LIN {X 0,Y 144.028,Z 768.399,A -85,B 0,C 180,E1 -24191.511,E2 -24191.511} C_VEL
LIN {X 0,Y 142.223,Z 772.01,A -85,B 0,C 180,E1 -24195.698,E2 -24195.698} C_VEL
LIN {X 0,Y 141.401,Z 773.873,A -85,B 0,C 180,E1 -24198.535,E2 -24198.535} C_VEL
LIN {X 0,Y 140.849,Z 775.271,A -85,B 0,C 180,E1 -24201.394,E2 -24201.394} C_VEL
LIN {X 0,Y 140.554,Z 776.27,A -85,B 0,C 180,E1 -24204.263,E2 -24204.263} C_VEL
LIN {X 0,Y 140.569,Z 777.067,A -85,B 0,C 180,E1 -24209.359,E2 -24209.359} C_VEL
LIN {X 0,Y 140.705,Z 776.87,A -85,B 0,C 180,E1 -24212.866,E2 -24212.866} C_VEL
LIN {X 0,Y 141.078,Z 776.256,A -85,B 0,C 180,E1 -24215.721,E2 -24215.721} C_VEL
LIN {X 0,Y 142.6,Z 773.851,A -85,B 0,C 180,E1 -24221.372,E2 -24221.372} C_VEL
LIN {X 0,Y 144.414,Z 771.718,A -85,B 0,C 180,E1 -24224.805,E2 -24224.805} C_VEL
LIN {X 0,Y 147.56,Z 777.302,A -85,B 0,C 180,E1 -24230.931,E2 -24230.931} C_VEL
LIN {X 0,Y 150.794,Z 779.846,A -85,B 0,C 180,E1 -24234.803,E2 -24234.803} C_VEL
LIN {X 0,Y 153.542,Z 781.108,A -85,B 0,C 180,E1 -24237.243,E2 -24237.243} C_VEL
LIN {X 0,Y 156.869,Z 781.934,A -85,B 0,C 180,E1 -24239.528,E2 -24239.528} C_VEL
LIN {X 0,Y 164.35,Z 782.268,A -85,B 0,C 180,E1 -24243.776,E2 -24243.776} C_VEL
LIN {X 0,Y 168.6,Z 781.872,A -85,B 0,C 180,E1 -24245.705,E2 -24245.705} C_VEL
LIN {X 0,Y 173.147,Z 780.97,A -85,B 0,C 180,E1 -24247.508,E2 -24247.508} C_VEL
LIN {X 0,Y 182.916,Z 777.866,A -85,B 0,C 180,E1 -24250.784,E2 -24250.784} C_VEL
LIN {X 0,Y 190.879,Z 774.269,A -85,B 0,C 180,E1 -24252.936,E2 -24252.936} C_VEL
LIN {X 0,Y 199.307,Z 769.471,A -85,B 0,C 180,E1 -24254.851,E2 -24254.851} C_VEL
LIN {X 0,Y 203.849,Z 766.375,A -85,B 0,C 180,E1 -24255.76,E2 -24255.76} C_VEL
LIN {X 0,Y 203.147,Z 766.886,A -85,B 0,C 180,E1 -24256.218,E2 -24256.218} C_VEL
LIN {X 0,Y 194.513,Z 772.435,A -85,B 0,C 180,E1 -24258.054,E2 -24258.054} C_VEL
LIN {X 0,Y 186.285,Z 776.45,A -85,B 0,C 180,E1 -24260.107,E2 -24260.107} C_VEL
LIN {X 0,Y 181.112,Z 778.475,A -85,B 0,C 180,E1 -24261.62,E2 -24261.62} C_VEL
LIN {X 0,Y 176.183,Z 779.958,A -85,B 0,C 180,E1 -24263.248,E2 -24263.248} C_VEL
LIN {X 0,Y 171.503,Z 780.907,A -85,B 0,C 180,E1 -24264.991,E2 -24264.991} C_VEL
LIN {X 0,Y 167.024,Z 781.435,A -85,B 0,C 180,E1 -24266.838,E2 -24266.838} C_VEL
LIN {X 0,Y 162.831,Z 781.546,A -85,B 0,C 180,E1 -24268.806,E2 -24268.806} C_VEL
LIN {X 0,Y 159.015,Z 781.191,A -85,B 0,C 180,E1 -24270.911,E2 -24270.911} C_VEL
LIN {X 0,Y 155.536,Z 780.325,A -85,B 0,C 180,E1 -24273.137,E2 -24273.137} C_VEL
LIN {X 0,Y 152.482,Z 779.046,A -85,B 0,C 180,E1 -24275.492,E2 -24275.492} C_VEL
LIN {X 0,Y 148.803,Z 776.375,A -85,B 0,C 180,E1 -24279.254,E2 -24279.254} C_VEL
LIN {X 0,Y 146.088,Z 772.671,A -85,B 0,C 180,E1 -24283.223,E2 -24283.223} C_VEL
LIN {X 0,Y 144.244,Z 767.118,A -85,B 0,C 180,E1 -24287.917,E2 -24287.917} C_VEL
LIN {X 0,Y 143.675,Z 760.498,A -85,B 0,C 180,E1 -24292.269,E2 -24292.269} C_VEL
LIN {X 0,Y 143.884,Z 753.954,A -85,B 0,C 180,E1 -24295.798,E2 -24295.798} C_VEL
LIN {X 0,Y 144.25,Z 747.49,A -85,B 0,C 180,E1 -24298.604,E2 -24298.604} C_VEL
LIN {X 0,Y 144.568,Z 738.067,A -85,B 0,C 180,E1 -24301.741,E2 -24301.741} C_VEL
LIN {X 0,Y 144.815,Z 730.254,A -85,B 0,C 180,E1 -24303.826,E2 -24303.826} C_VEL
LIN {X 0,Y 145.107,Z 718.487,A -85,B 0,C 180,E1 -24306.256,E2 -24306.256} C_VEL
LIN {X 0,Y 145.333,Z 708.147,A -85,B 0,C 180,E1 -24307.817,E2 -24307.817} C_VEL
LIN {X 0,Y 145.44,Z 690.055,A -85,B 0,C 180,E1 -24309.737,E2 -24309.737} C_VEL
LIN {X 0,Y 145.416,Z 656.523,A -85,B 0,C 180,E1 -24313.05,E2 -24313.05} C_VEL
LIN {X 0,Y 143.902,Z 632.91,A -85,B 0,C 180,E1 -24315.219,E2 -24315.219} C_VEL
LIN {X 0,Y 143.753,Z 627.443,A -85,B 0,C 180,E1 -24317.058,E2 -24317.058} C_VEL
LIN {X 0,Y 145.393,Z 608.667,A -85,B 0,C 180,E1 -24323.842,E2 -24323.842} C_VEL
LIN {X 0,Y 145.884,Z 605.68,A -85,B 0,C 180,E1 -24325.312,E2 -24325.312} C_VEL
LIN {X 0,Y 146.21,Z 605.142,A -85,B 0,C 180,E1 -24326.016,E2 -24326.016} C_VEL
LIN {X 0,Y 147.642,Z 604.988,A -85,B 0,C 180,E1 -24327.269,E2 -24327.269} C_VEL
LIN {X 0,Y 149.873,Z 603.29,A -85,B 0,C 180,E1 -24328.728,E2 -24328.728} C_VEL
LIN {X 0,Y 154.133,Z 597.997,A -85,B 0,C 180,E1 -24331.052,E2 -24331.052} C_VEL
LIN {X 0,Y 154.864,Z 597.508,A -85,B 0,C 180,E1 -24331.459,E2 -24331.459} C_VEL
LIN {X 0,Y 157.666,Z 597.465,A -85,B 0,C 180,E1 -24333.097,E2 -24333.097} C_VEL
LIN {X 0,Y 159.705,Z 596.432,A -85,B 0,C 180,E1 -24334.131,E2 -24334.131} C_VEL
LIN {X 0,Y 164.294,Z 595.958,A -85,B 0,C 180,E1 -24336.408,E2 -24336.408} C_VEL
LIN {X 0,Y 165.416,Z 595.863,A -85,B 0,C 180,E1 -24336.93,E2 -24336.93} C_VEL
LIN {X 0,Y 171.993,Z 606.336,A -85,B 0,C 180,E1 -24340.443,E2 -24340.443} C_VEL
LIN {X 0,Y 177.72,Z 616.812,A -85,B 0,C 180,E1 -24343.192,E2 -24343.192} C_VEL
LIN {X 0,Y 180.855,Z 624.587,A -85,B 0,C 180,E1 -24344.681,E2 -24344.681} C_VEL
LIN {X 0,Y 178.029,Z 666.301,A -85,B 0,C 180,E1 -24346.194,E2 -24346.194} C_VEL
LIN {X 0,Y 176.211,Z 679.252,A -85,B 0,C 180,E1 -24347.012,E2 -24347.012} C_VEL
LIN {X 0,Y 173.885,Z 691.223,A -85,B 0,C 180,E1 -24348.17,E2 -24348.17} C_VEL
LIN {X 0,Y 170.991,Z 702.495,A -85,B 0,C 180,E1 -24349.656,E2 -24349.656} C_VEL
LIN {X 0,Y 167.18,Z 714.119,A -85,B 0,C 180,E1 -24351.676,E2 -24351.676} C_VEL
LIN {X 0,Y 163.151,Z 724.561,A -85,B 0,C 180,E1 -24354.059,E2 -24354.059} C_VEL
LIN {X 0,Y 159.522,Z 733.089,A -85,B 0,C 180,E1 -24356.584,E2 -24356.584} C_VEL
LIN {X 0,Y 155.782,Z 741.183,A -85,B 0,C 180,E1 -24359.624,E2 -24359.624} C_VEL
LIN {X 0,Y 151.851,Z 748.611,A -85,B 0,C 180,E1 -24363.173,E2 -24363.173} C_VEL
LIN {X 0,Y 147.83,Z 755.661,A -85,B 0,C 180,E1 -24367.643,E2 -24367.643} C_VEL
LIN {X 0,Y 145.189,Z 760.348,A -85,B 0,C 180,E1 -24371.659,E2 -24371.659} C_VEL
LIN {X 0,Y 143.132,Z 763.929,A -85,B 0,C 180,E1 -24375.786,E2 -24375.786} C_VEL
LIN {X 0,Y 142.14,Z 765.777,A -85,B 0,C 180,E1 -24378.59,E2 -24378.59} C_VEL
LIN {X 0,Y 141.435,Z 767.165,A -85,B 0,C 180,E1 -24381.424,E2 -24381.424} C_VEL
LIN {X 0,Y 141.008,Z 768.151,A -85,B 0,C 180,E1 -24384.277,E2 -24384.277} C_VEL
LIN {X 0,Y 140.737,Z 768.758,A -85,B 0,C 180,E1 -24387.135,E2 -24387.135} C_VEL
LIN {X 0,Y 140.69,Z 768.984,A -85,B 0,C 180,E1 -24389.997,E2 -24389.997} C_VEL
LIN {X 0,Y 140.736,Z 768.789,A -85,B 0,C 180,E1 -24392.86,E2 -24392.86} C_VEL
LIN {X 0,Y 141.007,Z 768.204,A -85,B 0,C 180,E1 -24395.718,E2 -24395.718} C_VEL
LIN {X 0,Y 142.136,Z 765.884,A -85,B 0,C 180,E1 -24401.405,E2 -24401.405} C_VEL
LIN {X 0,Y 143.73,Z 763.013,A -85,B 0,C 180,E1 -24405.598,E2 -24405.598} C_VEL
LIN {X 0,Y 145.977,Z 759.117,A -85,B 0,C 180,E1 -24409.692,E2 -24409.692} C_VEL
LIN {X 0,Y 148.832,Z 754.096,A -85,B 0,C 180,E1 -24413.662,E2 -24413.662} C_VEL
LIN {X 0,Y 152.426,Z 747.763,A -85,B 0,C 180,E1 -24417.454,E2 -24417.454} C_VEL
LIN {X 0,Y 156.142,Z 740.567,A -85,B 0,C 180,E1 -24420.801,E2 -24420.801} C_VEL
LIN {X 0,Y 160.208,Z 731.769,A -85,B 0,C 180,E1 -24424.005,E2 -24424.005} C_VEL
LIN {X 0,Y 164.355,Z 721.911,A -85,B 0,C 180,E1 -24426.771,E2 -24426.771} C_VEL
LIN {X 0,Y 168.491,Z 710.804,A -85,B 0,C 180,E1 -24429.112,E2 -24429.112} C_VEL
LIN {X 0,Y 171.827,Z 699.911,A -85,B 0,C 180,E1 -24430.873,E2 -24430.873} C_VEL
LIN {X 0,Y 174.767,Z 687.858,A -85,B 0,C 180,E1 -24432.341,E2 -24432.341} C_VEL
LIN {X 0,Y 177.064,Z 675.297,A -85,B 0,C 180,E1 -24433.417,E2 -24433.417} C_VEL
LIN {X 0,Y 178.617,Z 661.534,A -85,B 0,C 180,E1 -24434.161,E2 -24434.161} C_VEL
LIN {X 0,Y 181.017,Z 624.783,A -85,B 0,C 180,E1 -24435.451,E2 -24435.451} C_VEL
LIN {X 0,Y 177.262,Z 615.771,A -85,B 0,C 180,E1 -24437.232,E2 -24437.232} C_VEL
LIN {X 0,Y 171.653,Z 605.747,A -85,B 0,C 180,E1 -24439.947,E2 -24439.947} C_VEL
LIN {X 0,Y 166.095,Z 596.95,A -85,B 0,C 180,E1 -24442.917,E2 -24442.917} C_VEL
LIN {X 0,Y 161.752,Z 590.626,A -85,B 0,C 180,E1 -24445.502,E2 -24445.502} C_VEL
LIN {X 0,Y 159.087,Z 586.943,A -85,B 0,C 180,E1 -24447.236,E2 -24447.236} C_VEL
LIN {X 0,Y 156.431,Z 583.247,A -85,B 0,C 180,E1 -24449.115,E2 -24449.115} C_VEL
LIN {X 0,Y 153.386,Z 579.693,A -85,B 0,C 180,E1 -24451.429,E2 -24451.429} C_VEL
LIN {X 0,Y 152.306,Z 577.95,A -85,B 0,C 180,E1 -24452.364,E2 -24452.364} C_VEL
LIN {X 0,Y 149.696,Z 575.629,A -85,B 0,C 180,E1 -24454.609,E2 -24454.609} C_VEL
LIN {X 0,Y 148.169,Z 572.836,A -85,B 0,C 180,E1 -24456.223,E2 -24456.223} C_VEL
LIN {X 0,Y 147.867,Z 572.413,A -85,B 0,C 180,E1 -24456.543,E2 -24456.543} C_VEL
LIN {X 0,Y 145.469,Z 570.904,A -85,B 0,C 180,E1 -24459.052,E2 -24459.052} C_VEL
LIN {X 0,Y 143.832,Z 568.536,A -85,B 0,C 180,E1 -24461.205,E2 -24461.205} C_VEL
LIN {X 0,Y 143.277,Z 566.62,A -85,B 0,C 180,E1 -24462.331,E2 -24462.331} C_VEL
LIN {X 0,Y 143.588,Z 566.58,A -85,B 0,C 180,E1 -24468.709,E2 -24468.709} C_VEL
LIN {X 0,Y 143.658,Z 566.571,A -85,B 0,C 180,E1 -24471.56,E2 -24471.56} C_VEL
LIN {X 0,Y 144.172,Z 566.526,A -85,B 0,C 180,E1 -24480,E2 -24480} C_VEL
LIN {X 0,Y 143.678,Z 566.573,A -85,B 0,C 180,E1 -24488.438,E2 -24488.438} C_VEL
LIN {X 0,Y 143.565,Z 566.586,A -85,B 0,C 180,E1 -24491.758,E2 -24491.758} C_VEL
LIN {X 0,Y 143.287,Z 566.712,A -85,B 0,C 180,E1 -24497.483,E2 -24497.483} C_VEL
LIN {X 0,Y 143.993,Z 568.912,A -85,B 0,C 180,E1 -24498.681,E2 -24498.681} C_VEL
LIN {X 0,Y 145.834,Z 571.244,A -85,B 0,C 180,E1 -24501.008,E2 -24501.008} C_VEL
LIN {X 0,Y 148.092,Z 572.648,A -85,B 0,C 180,E1 -24503.326,E2 -24503.326} C_VEL
LIN {X 0,Y 149.662,Z 575.61,A -85,B 0,C 180,E1 -24505.001,E2 -24505.001} C_VEL
LIN {X 0,Y 152.591,Z 578.318,A -85,B 0,C 180,E1 -24507.517,E2 -24507.517} C_VEL
LIN {X 0,Y 154.86,Z 581.681,A -85,B 0,C 180,E1 -24509.387,E2 -24509.387} C_VEL
LIN {X 0,Y 156.547,Z 583.503,A -85,B 0,C 180,E1 -24510.618,E2 -24510.618} C_VEL
LIN {X 0,Y 159.281,Z 587.171,A -85,B 0,C 180,E1 -24512.531,E2 -24512.531} C_VEL
LIN {X 0,Y 161.27,Z 590.154,A -85,B 0,C 180,E1 -24513.848,E2 -24513.848} C_VEL
LIN {X 0,Y 165.359,Z 596.983,A -85,B 0,C 180,E1 -24516.384,E2 -24516.384} C_VEL
LIN {X 0,Y 170.544,Z 606.854,A -85,B 0,C 180,E1 -24519.316,E2 -24519.316} C_VEL
LIN {X 0,Y 175.217,Z 617.057,A -85,B 0,C 180,E1 -24521.752,E2 -24521.752} C_VEL
LIN {X 0,Y 179.914,Z 629.167,A -85,B 0,C 180,E1 -24524.074,E2 -24524.074} C_VEL
LIN {X 0,Y 180.657,Z 631.54,A -85,B 0,C 180,E1 -24524.447,E2 -24524.447} C_VEL
LIN {X 0,Y 177.79,Z 673.247,A -85,B 0,C 180,E1 -24525.933,E2 -24525.933} C_VEL
LIN {X 0,Y 175.882,Z 686.736,A -85,B 0,C 180,E1 -24526.773,E2 -24526.773} C_VEL
LIN {X 0,Y 173.121,Z 699.519,A -85,B 0,C 180,E1 -24527.949,E2 -24527.949} C_VEL
LIN {X 0,Y 170.042,Z 710.602,A -85,B 0,C 180,E1 -24529.389,E2 -24529.389} C_VEL
LIN {X 0,Y 166.132,Z 722.153,A -85,B 0,C 180,E1 -24531.396,E2 -24531.396} C_VEL
LIN {X 0,Y 162.027,Z 732.557,A -85,B 0,C 180,E1 -24533.776,E2 -24533.776} C_VEL
LIN {X 0,Y 158.192,Z 741.068,A -85,B 0,C 180,E1 -24536.269,E2 -24536.269} C_VEL
LIN {X 0,Y 154.4,Z 748.922,A -85,B 0,C 180,E1 -24539.201,E2 -24539.201} C_VEL
LIN {X 0,Y 150.544,Z 756.602,A -85,B 0,C 180,E1 -24542.927,E2 -24542.927} C_VEL
LIN {X 0,Y 147.137,Z 762.745,A -85,B 0,C 180,E1 -24546.772,E2 -24546.772} C_VEL
LIN {X 0,Y 145.111,Z 765.37,A -85,B 0,C 180,E1 -24548.7,E2 -24548.7} C_VEL
LIN {X 0,Y 140.306,Z 769.068,A -85,B 0,C 180,E1 -24551.862,E2 -24551.862} C_VEL
LIN {X 0,Y 136.608,Z 771.488,A -85,B 0,C 180,E1 -24554.599,E2 -24554.599} C_VEL
LIN {X 0,Y 134.793,Z 773.041,A -85,B 0,C 180,E1 -24556.879,E2 -24556.879} C_VEL
LIN {X 0,Y 134.497,Z 773.51,A -85,B 0,C 180,E1 -24557.678,E2 -24557.678} C_VEL
LIN {X 0,Y 133.823,Z 775.066,A -85,B 0,C 180,E1 -24560.938,E2 -24560.938} C_VEL
LIN {X 0,Y 133.397,Z 776.676,A -85,B 0,C 180,E1 -24566.983,E2 -24566.983} C_VEL
LIN {X 0,Y 133.532,Z 776.891,A -85,B 0,C 180,E1 -24570.003,E2 -24570.003} C_VEL
LIN {X 0,Y 134.028,Z 776.052,A -85,B 0,C 180,E1 -24576.023,E2 -24576.023} C_VEL
LIN {X 0,Y 135.653,Z 773.646,A -85,B 0,C 180,E1 -24581.963,E2 -24581.963} C_VEL
LIN {X 0,Y 138.304,Z 770.641,A -85,B 0,C 180,E1 -24586.611,E2 -24586.611} C_VEL
LIN {X 0,Y 141.148,Z 775.592,A -85,B 0,C 180,E1 -24591.93,E2 -24591.93} C_VEL
LIN {X 0,Y 144.491,Z 778.609,A -85,B 0,C 180,E1 -24595.963,E2 -24595.963} C_VEL
LIN {X 0,Y 147.354,Z 780.07,A -85,B 0,C 180,E1 -24598.489,E2 -24598.489} C_VEL
LIN {X 0,Y 154.444,Z 781.964,A -85,B 0,C 180,E1 -24603.1,E2 -24603.1} C_VEL
LIN {X 0,Y 158.507,Z 782.227,A -85,B 0,C 180,E1 -24605.201,E2 -24605.201} C_VEL
LIN {X 0,Y 162.885,Z 782.108,A -85,B 0,C 180,E1 -24607.163,E2 -24607.163} C_VEL
LIN {X 0,Y 167.589,Z 781.623,A -85,B 0,C 180,E1 -24608.982,E2 -24608.982} C_VEL
LIN {X 0,Y 172.532,Z 780.703,A -85,B 0,C 180,E1 -24610.676,E2 -24610.676} C_VEL
LIN {X 0,Y 177.661,Z 779.286,A -85,B 0,C 180,E1 -24612.262,E2 -24612.262} C_VEL
LIN {X 0,Y 185.853,Z 776.369,A -85,B 0,C 180,E1 -24614.395,E2 -24614.395} C_VEL
LIN {X 0,Y 189.989,Z 774.505,A -85,B 0,C 180,E1 -24615.344,E2 -24615.344} C_VEL
LIN {X 0,Y 192.289,Z 773.406,A -85,B 0,C 180,E1 -24616.018,E2 -24616.018} C_VEL
LIN {X 0,Y 183.718,Z 777.157,A -85,B 0,C 180,E1 -24617.975,E2 -24617.975} C_VEL
LIN {X 0,Y 175.648,Z 779.743,A -85,B 0,C 180,E1 -24620.194,E2 -24620.194} C_VEL
LIN {X 0,Y 166.894,Z 781.396,A -85,B 0,C 180,E1 -24623.143,E2 -24623.143} C_VEL
LIN {X 0,Y 161.119,Z 781.691,A -85,B 0,C 180,E1 -24625.455,E2 -24625.455} C_VEL
LIN {X 0,Y 156.808,Z 781.382,A -85,B 0,C 180,E1 -24627.464,E2 -24627.464} C_VEL
LIN {X 0,Y 152.879,Z 780.647,A -85,B 0,C 180,E1 -24629.623,E2 -24629.623} C_VEL
LIN {X 0,Y 149.294,Z 779.53,A -85,B 0,C 180,E1 -24631.917,E2 -24631.917} C_VEL
LIN {X 0,Y 144.767,Z 777.023,A -85,B 0,C 180,E1 -24635.629,E2 -24635.629} C_VEL
LIN {X 0,Y 141.32,Z 773.548,A -85,B 0,C 180,E1 -24639.628,E2 -24639.628} C_VEL
LIN {X 0,Y 138.685,Z 768.495,A -85,B 0,C 180,E1 -24644.341,E2 -24644.341} C_VEL
LIN {X 0,Y 137.443,Z 762.266,A -85,B 0,C 180,E1 -24648.945,E2 -24648.945} C_VEL
LIN {X 0,Y 137.312,Z 756.216,A -85,B 0,C 180,E1 -24652.649,E2 -24652.649} C_VEL
LIN {X 0,Y 137.636,Z 748.736,A -85,B 0,C 180,E1 -24656.341,E2 -24656.341} C_VEL
LIN {X 0,Y 137.901,Z 741.278,A -85,B 0,C 180,E1 -24659.27,E2 -24659.27} C_VEL
LIN {X 0,Y 138.187,Z 733.012,A -85,B 0,C 180,E1 -24661.822,E2 -24661.822} C_VEL
LIN {X 0,Y 138.339,Z 723.891,A -85,B 0,C 180,E1 -24664.006,E2 -24664.006} C_VEL
LIN {X 0,Y 138.591,Z 713.294,A -85,B 0,C 180,E1 -24666.004,E2 -24666.004} C_VEL
LIN {X 0,Y 138.742,Z 700.731,A -85,B 0,C 180,E1 -24667.641,E2 -24667.641} C_VEL
LIN {X 0,Y 138.647,Z 657.852,A -85,B 0,C 180,E1 -24672.236,E2 -24672.236} C_VEL
LIN {X 0,Y 136.908,Z 632.582,A -85,B 0,C 180,E1 -24674.7,E2 -24674.7} C_VEL
LIN {X 0,Y 136.728,Z 626.035,A -85,B 0,C 180,E1 -24677.191,E2 -24677.191} C_VEL
LIN {X 0,Y 137.028,Z 622.984,A -85,B 0,C 180,E1 -24678.891,E2 -24678.891} C_VEL
LIN {X 0,Y 137.175,Z 622.556,A -85,B 0,C 180,E1 -24679.452,E2 -24679.452} C_VEL
LIN {X 0,Y 138.377,Z 622.348,A -85,B 0,C 180,E1 -24681.015,E2 -24681.015} C_VEL
LIN {X 0,Y 140.519,Z 619.897,A -85,B 0,C 180,E1 -24682.889,E2 -24682.889} C_VEL
LIN {X 0,Y 145.658,Z 612.31,A -85,B 0,C 180,E1 -24686.508,E2 -24686.508} C_VEL
LIN {X 0,Y 148.347,Z 611.466,A -85,B 0,C 180,E1 -24688.454,E2 -24688.454} C_VEL
LIN {X 0,Y 151.116,Z 609.222,A -85,B 0,C 180,E1 -24690.143,E2 -24690.143} C_VEL
LIN {X 0,Y 155.04,Z 604.642,A -85,B 0,C 180,E1 -24692.184,E2 -24692.184} C_VEL
LIN {X 0,Y 157.427,Z 604.468,A -85,B 0,C 180,E1 -24693.536,E2 -24693.536} C_VEL
LIN {X 0,Y 159.975,Z 603.536,A -85,B 0,C 180,E1 -24694.828,E2 -24694.828} C_VEL
LIN {X 0,Y 163.435,Z 603.345,A -85,B 0,C 180,E1 -24696.535,E2 -24696.535} C_VEL
LIN {X 0,Y 168.981,Z 612.485,A -85,B 0,C 180,E1 -24699.625,E2 -24699.625} C_VEL
LIN {X 0,Y 173.751,Z 621.62,A -85,B 0,C 180,E1 -24702.06,E2 -24702.06} C_VEL
LIN {X 0,Y 175.803,Z 626.867,A -85,B 0,C 180,E1 -24703.112,E2 -24703.112} C_VEL
LIN {X 0,Y 172.998,Z 666.342,A -85,B 0,C 180,E1 -24704.558,E2 -24704.558} C_VEL
LIN {X 0,Y 171.072,Z 679.645,A -85,B 0,C 180,E1 -24705.41,E2 -24705.41} C_VEL
LIN {X 0,Y 168.411,Z 692.512,A -85,B 0,C 180,E1 -24706.686,E2 -24706.686} C_VEL
LIN {X 0,Y 165.161,Z 704.285,A -85,B 0,C 180,E1 -24708.324,E2 -24708.324} C_VEL
LIN {X 0,Y 161.198,Z 715.615,A -85,B 0,C 180,E1 -24710.382,E2 -24710.382} C_VEL
LIN {X 0,Y 157.04,Z 725.823,A -85,B 0,C 180,E1 -24712.829,E2 -24712.829} C_VEL
LIN {X 0,Y 152.807,Z 734.979,A -85,B 0,C 180,E1 -24715.706,E2 -24715.706} C_VEL
LIN {X 0,Y 148.332,Z 743.875,A -85,B 0,C 180,E1 -24719.378,E2 -24719.378} C_VEL
LIN {X 0,Y 144.284,Z 751.036,A -85,B 0,C 180,E1 -24723.218,E2 -24723.218} C_VEL
LIN {X 0,Y 141.28,Z 755.868,A -85,B 0,C 180,E1 -24726.547,E2 -24726.547} C_VEL
LIN {X 0,Y 138.469,Z 760.554,A -85,B 0,C 180,E1 -24730.734,E2 -24730.734} C_VEL
LIN {X 0,Y 136.246,Z 764.135,A -85,B 0,C 180,E1 -24735.051,E2 -24735.051} C_VEL
LIN {X 0,Y 135.175,Z 765.983,A -85,B 0,C 180,E1 -24737.994,E2 -24737.994} C_VEL
LIN {X 0,Y 134.429,Z 767.369,A -85,B 0,C 180,E1 -24740.974,E2 -24740.974} C_VEL
LIN {X 0,Y 133.95,Z 768.356,A -85,B 0,C 180,E1 -24743.974,E2 -24743.974} C_VEL
LIN {X 0,Y 133.596,Z 769.099,A -85,B 0,C 180,E1 -24748.24,E2 -24748.24} C_VEL
LIN {X 0,Y 133.659,Z 768.993,A -85,B 0,C 180,E1 -24753.011,E2 -24753.011} C_VEL
LIN {X 0,Y 133.948,Z 768.409,A -85,B 0,C 180,E1 -24756.021,E2 -24756.021} C_VEL
LIN {X 0,Y 135.171,Z 766.089,A -85,B 0,C 180,E1 -24762.001,E2 -24762.001} C_VEL
LIN {X 0,Y 136.901,Z 763.217,A -85,B 0,C 180,E1 -24766.398,E2 -24766.398} C_VEL
LIN {X 0,Y 139.306,Z 759.321,A -85,B 0,C 180,E1 -24770.677,E2 -24770.677} C_VEL
LIN {X 0,Y 142.347,Z 754.299,A -85,B 0,C 180,E1 -24774.81,E2 -24774.81} C_VEL
LIN {X 0,Y 146.163,Z 747.966,A -85,B 0,C 180,E1 -24778.737,E2 -24778.737} C_VEL
LIN {X 0,Y 150.678,Z 739.542,A -85,B 0,C 180,E1 -24782.705,E2 -24782.705} C_VEL
LIN {X 0,Y 155.218,Z 730.194,A -85,B 0,C 180,E1 -24786.056,E2 -24786.056} C_VEL
LIN {X 0,Y 159.665,Z 719.838,A -85,B 0,C 180,E1 -24788.844,E2 -24788.844} C_VEL
LIN {X 0,Y 164.043,Z 708.159,A -85,B 0,C 180,E1 -24791.198,E2 -24791.198} C_VEL
LIN {X 0,Y 167.56,Z 696.486,A -85,B 0,C 180,E1 -24792.964,E2 -24792.964} C_VEL
LIN {X 0,Y 170.383,Z 684.338,A -85,B 0,C 180,E1 -24794.315,E2 -24794.315} C_VEL
LIN {X 0,Y 172.602,Z 671.307,A -85,B 0,C 180,E1 -24795.308,E2 -24795.308} C_VEL
LIN {X 0,Y 173.916,Z 657.301,A -85,B 0,C 180,E1 -24795.964,E2 -24795.964} C_VEL
LIN {X 0,Y 175.972,Z 627.04,A -85,B 0,C 180,E1 -24797.024,E2 -24797.024} C_VEL
LIN {X 0,Y 172.81,Z 619.484,A -85,B 0,C 180,E1 -24798.633,E2 -24798.633} C_VEL
LIN {X 0,Y 167.634,Z 610.173,A -85,B 0,C 180,E1 -24801.322,E2 -24801.322} C_VEL
LIN {X 0,Y 162.011,Z 600.921,A -85,B 0,C 180,E1 -24804.586,E2 -24804.586} C_VEL
LIN {X 0,Y 156.679,Z 593.19,A -85,B 0,C 180,E1 -24808.103,E2 -24808.103} C_VEL
LIN {X 0,Y 153.194,Z 588.56,A -85,B 0,C 180,E1 -24810.714,E2 -24810.714} C_VEL
LIN {X 0,Y 150.501,Z 584.839,A -85,B 0,C 180,E1 -24812.995,E2 -24812.995} C_VEL
LIN {X 0,Y 147.145,Z 581.167,A -85,B 0,C 180,E1 -24816.141,E2 -24816.141} C_VEL
LIN {X 0,Y 146.081,Z 579.156,A -85,B 0,C 180,E1 -24817.363,E2 -24817.363} C_VEL
LIN {X 0,Y 143.353,Z 576.977,A -85,B 0,C 180,E1 -24820.489,E2 -24820.489} C_VEL
LIN {X 0,Y 141.734,Z 573.899,A -85,B 0,C 180,E1 -24822.97,E2 -24822.97} C_VEL
LIN {X 0,Y 141.469,Z 573.476,A -85,B 0,C 180,E1 -24823.402,E2 -24823.402} C_VEL
LIN {X 0,Y 138.7,Z 571.786,A -85,B 0,C 180,E1 -24828.306,E2 -24828.306} C_VEL
LIN {X 0,Y 136.736,Z 568.099,A -85,B 0,C 180,E1 -24835.578,E2 -24835.578} C_VEL
LIN {X 0,Y 136.722,Z 567.429,A -85,B 0,C 180,E1 -24836.685,E2 -24836.685} C_VEL
LIN {X 0,Y 137.129,Z 567.403,A -85,B 0,C 180,E1 -24840,E2 -24840} C_VEL
LIN {X 0,Y 136.712,Z 567.539,A -85,B 0,C 180,E1 -24843.5,E2 -24843.5} C_VEL
LIN {X 0,Y 137.235,Z 569.712,A -85,B 0,C 180,E1 -24846.986,E2 -24846.986} C_VEL
LIN {X 0,Y 140.336,Z 573.047,A -85,B 0,C 180,E1 -24854.501,E2 -24854.501} C_VEL
LIN {X 0,Y 141.681,Z 573.747,A -85,B 0,C 180,E1 -24856.572,E2 -24856.572} C_VEL
LIN {X 0,Y 143.097,Z 576.625,A -85,B 0,C 180,E1 -24858.803,E2 -24858.803} C_VEL
LIN {X 0,Y 145.486,Z 578.849,A -85,B 0,C 180,E1 -24861.663,E2 -24861.663} C_VEL
LIN {X 0,Y 146.238,Z 579.437,A -85,B 0,C 180,E1 -24862.46,E2 -24862.46} C_VEL
LIN {X 0,Y 148.311,Z 582.736,A -85,B 0,C 180,E1 -24864.683,E2 -24864.683} C_VEL
LIN {X 0,Y 150.439,Z 584.807,A -85,B 0,C 180,E1 -24866.594,E2 -24866.594} C_VEL
LIN {X 0,Y 153.062,Z 588.426,A -85,B 0,C 180,E1 -24868.824,E2 -24868.824} C_VEL
LIN {X 0,Y 154.391,Z 590.164,A -85,B 0,C 180,E1 -24869.86,E2 -24869.86} C_VEL
LIN {X 0,Y 157.717,Z 594.697,A -85,B 0,C 180,E1 -24872.267,E2 -24872.267} C_VEL
LIN {X 0,Y 162.367,Z 602.859,A -85,B 0,C 180,E1 -24875.376,E2 -24875.376} C_VEL
LIN {X 0,Y 167.211,Z 612.47,A -85,B 0,C 180,E1 -24878.291,E2 -24878.291} C_VEL
LIN {X 0,Y 171.382,Z 622.025,A -85,B 0,C 180,E1 -24880.617,E2 -24880.617} C_VEL
LIN {X 0,Y 175.614,Z 633.499,A -85,B 0,C 180,E1 -24882.87,E2 -24882.87} C_VEL
LIN {X 0,Y 172.714,Z 673.501,A -85,B 0,C 180,E1 -24884.321,E2 -24884.321} C_VEL
LIN {X 0,Y 170.734,Z 686.804,A -85,B 0,C 180,E1 -24885.163,E2 -24885.163} C_VEL
LIN {X 0,Y 167.93,Z 699.322,A -85,B 0,C 180,E1 -24886.331,E2 -24886.331} C_VEL
LIN {X 0,Y 164.716,Z 710.402,A -85,B 0,C 180,E1 -24887.781,E2 -24887.781} C_VEL
LIN {X 0,Y 160.625,Z 721.951,A -85,B 0,C 180,E1 -24889.81,E2 -24889.81} C_VEL
LIN {X 0,Y 156.337,Z 732.355,A -85,B 0,C 180,E1 -24892.233,E2 -24892.233} C_VEL
LIN {X 0,Y 152.333,Z 740.866,A -85,B 0,C 180,E1 -24894.785,E2 -24894.785} C_VEL
LIN {X 0,Y 148.323,Z 748.719,A -85,B 0,C 180,E1 -24897.791,E2 -24897.791} C_VEL
LIN {X 0,Y 144.216,Z 756.4,A -85,B 0,C 180,E1 -24901.636,E2 -24901.636} C_VEL
LIN {X 0,Y 140.066,Z 763.48,A -85,B 0,C 180,E1 -24906.337,E2 -24906.337} C_VEL
LIN {X 0,Y 137.28,Z 768.194,A -85,B 0,C 180,E1 -24910.566,E2 -24910.566} C_VEL
LIN {X 0,Y 135.33,Z 771.806,A -85,B 0,C 180,E1 -24914.953,E2 -24914.953} C_VEL
LIN {X 0,Y 134.497,Z 773.51,A -85,B 0,C 180,E1 -24917.678,E2 -24917.678} C_VEL
LIN {X 0,Y 133.339,Z 774.824,A -85,B 0,C 180,E1 -24920.089,E2 -24920.089} C_VEL
LIN {X 0,Y 131.45,Z 775.762,A -85,B 0,C 180,E1 -24922.493,E2 -24922.493} C_VEL
LIN {X 0,Y 127.514,Z 776.645,A -85,B 0,C 180,E1 -24927.488,E2 -24927.488} C_VEL
LIN {X 0,Y 126.493,Z 776.685,A -85,B 0,C 180,E1 -24930.147,E2 -24930.147} C_VEL
LIN {X 0,Y 126.427,Z 776.612,A -85,B 0,C 180,E1 -24931.049,E2 -24931.049} C_VEL
LIN {X 0,Y 126.974,Z 775.847,A -85,B 0,C 180,E1 -24936.358,E2 -24936.358} C_VEL
LIN {X 0,Y 128.736,Z 773.441,A -85,B 0,C 180,E1 -24942.616,E2 -24942.616} C_VEL
LIN {X 0,Y 132.057,Z 769.625,A -85,B 0,C 180,E1 -24948.223,E2 -24948.223} C_VEL
LIN {X 0,Y 132.594,Z 769.669,A -85,B 0,C 180,E1 -24948.947,E2 -24948.947} C_VEL
LIN {X 0,Y 135.91,Z 774.849,A -85,B 0,C 180,E1 -24954.439,E2 -24954.439} C_VEL
LIN {X 0,Y 138.314,Z 777.034,A -85,B 0,C 180,E1 -24957.216,E2 -24957.216} C_VEL
LIN {X 0,Y 141.262,Z 778.863,A -85,B 0,C 180,E1 -24959.838,E2 -24959.838} C_VEL
LIN {X 0,Y 148.578,Z 781.249,A -85,B 0,C 180,E1 -24964.587,E2 -24964.587} C_VEL
LIN {X 0,Y 152.772,Z 781.931,A -85,B 0,C 180,E1 -24966.732,E2 -24966.732} C_VEL
LIN {X 0,Y 157.282,Z 782.168,A -85,B 0,C 180,E1 -24968.727,E2 -24968.727} C_VEL
LIN {X 0,Y 167.228,Z 781.399,A -85,B 0,C 180,E1 -24972.257,E2 -24972.257} C_VEL
LIN {X 0,Y 172.524,Z 780.446,A -85,B 0,C 180,E1 -24973.832,E2 -24973.832} C_VEL
LIN {X 0,Y 179.267,Z 778.665,A -85,B 0,C 180,E1 -24975.577,E2 -24975.577} C_VEL
LIN {X 0,Y 179.892,Z 778.469,A -85,B 0,C 180,E1 -24976.139,E2 -24976.139} C_VEL
LIN {X 0,Y 170.268,Z 780.755,A -85,B 0,C 180,E1 -24978.668,E2 -24978.668} C_VEL
LIN {X 0,Y 161.946,Z 781.672,A -85,B 0,C 180,E1 -24981.369,E2 -24981.369} C_VEL
LIN {X 0,Y 155.33,Z 781.545,A -85,B 0,C 180,E1 -24983.971,E2 -24983.971} C_VEL
LIN {X 0,Y 150.887,Z 780.937,A -85,B 0,C 180,E1 -24986.018,E2 -24986.018} C_VEL
LIN {X 0,Y 146.832,Z 779.963,A -85,B 0,C 180,E1 -24988.23,E2 -24988.23} C_VEL
LIN {X 0,Y 143.155,Z 778.487,A -85,B 0,C 180,E1 -24990.598,E2 -24990.598} C_VEL
LIN {X 0,Y 138.482,Z 775.553,A -85,B 0,C 180,E1 -24994.445,E2 -24994.445} C_VEL
LIN {X 0,Y 134.94,Z 771.629,A -85,B 0,C 180,E1 -24998.619,E2 -24998.619} C_VEL
LIN {X 0,Y 132.299,Z 765.976,A -85,B 0,C 180,E1 -25003.564,E2 -25003.564} C_VEL
LIN {X 0,Y 131.181,Z 760.426,A -85,B 0,C 180,E1 -25007.626,E2 -25007.626} C_VEL
LIN {X 0,Y 130.999,Z 752.827,A -85,B 0,C 180,E1 -25012.292,E2 -25012.292} C_VEL
LIN {X 0,Y 131.276,Z 746.503,A -85,B 0,C 180,E1 -25015.394,E2 -25015.394} C_VEL
LIN {X 0,Y 131.592,Z 738.567,A -85,B 0,C 180,E1 -25018.47,E2 -25018.47} C_VEL
LIN {X 0,Y 131.776,Z 729.84,A -85,B 0,C 180,E1 -25021.146,E2 -25021.146} C_VEL
LIN {X 0,Y 131.928,Z 718.356,A -85,B 0,C 180,E1 -25023.818,E2 -25023.818} C_VEL
LIN {X 0,Y 132.117,Z 708.986,A -85,B 0,C 180,E1 -25025.437,E2 -25025.437} C_VEL
LIN {X 0,Y 132.078,Z 691.697,A -85,B 0,C 180,E1 -25027.549,E2 -25027.549} C_VEL
LIN {X 0,Y 131.787,Z 657.243,A -85,B 0,C 180,E1 -25031.439,E2 -25031.439} C_VEL
LIN {X 0,Y 130.977,Z 648.915,A -85,B 0,C 180,E1 -25032.394,E2 -25032.394} C_VEL
LIN {X 0,Y 130.574,Z 645.694,A -85,B 0,C 180,E1 -25033.081,E2 -25033.081} C_VEL
LIN {X 0,Y 130.445,Z 644.215,A -85,B 0,C 180,E1 -25033.756,E2 -25033.756} C_VEL
LIN {X 0,Y 131.039,Z 643.587,A -85,B 0,C 180,E1 -25034.908,E2 -25034.908} C_VEL
LIN {X 0,Y 131.937,Z 641.098,A -85,B 0,C 180,E1 -25035.843,E2 -25035.843} C_VEL
LIN {X 0,Y 133.521,Z 635.471,A -85,B 0,C 180,E1 -25037.124,E2 -25037.124} C_VEL
LIN {X 0,Y 136.468,Z 629.724,A -85,B 0,C 180,E1 -25039.949,E2 -25039.949} C_VEL
LIN {X 0,Y 138.512,Z 628.96,A -85,B 0,C 180,E1 -25042.082,E2 -25042.082} C_VEL
LIN {X 0,Y 141.021,Z 626.277,A -85,B 0,C 180,E1 -25044.17,E2 -25044.17} C_VEL
LIN {X 0,Y 144.928,Z 620.747,A -85,B 0,C 180,E1 -25046.846,E2 -25046.846} C_VEL
LIN {X 0,Y 146.094,Z 619.191,A -85,B 0,C 180,E1 -25047.582,E2 -25047.582} C_VEL
LIN {X 0,Y 148.995,Z 617.996,A -85,B 0,C 180,E1 -25049.55,E2 -25049.55} C_VEL
LIN {X 0,Y 152.447,Z 615.153,A -85,B 0,C 180,E1 -25051.531,E2 -25051.531} C_VEL
LIN {X 0,Y 155.723,Z 611.722,A -85,B 0,C 180,E1 -25053.177,E2 -25053.177} C_VEL
LIN {X 0,Y 161.313,Z 610.411,A -85,B 0,C 180,E1 -25056.027,E2 -25056.027} C_VEL
LIN {X 0,Y 167.124,Z 620.791,A -85,B 0,C 180,E1 -25059.4,E2 -25059.4} C_VEL
LIN {X 0,Y 170.187,Z 627.288,A -85,B 0,C 180,E1 -25061.061,E2 -25061.061} C_VEL
LIN {X 0,Y 170.887,Z 629.16,A -85,B 0,C 180,E1 -25061.449,E2 -25061.449} C_VEL
LIN {X 0,Y 168.091,Z 666.648,A -85,B 0,C 180,E1 -25062.841,E2 -25062.841} C_VEL
LIN {X 0,Y 166.072,Z 680.048,A -85,B 0,C 180,E1 -25063.71,E2 -25063.71} C_VEL
LIN {X 0,Y 163.334,Z 692.723,A -85,B 0,C 180,E1 -25064.983,E2 -25064.983} C_VEL
LIN {X 0,Y 159.945,Z 704.494,A -85,B 0,C 180,E1 -25066.639,E2 -25066.639} C_VEL
LIN {X 0,Y 155.803,Z 715.824,A -85,B 0,C 180,E1 -25068.72,E2 -25068.72} C_VEL
LIN {X 0,Y 151.43,Z 726.031,A -85,B 0,C 180,E1 -25071.201,E2 -25071.201} C_VEL
LIN {X 0,Y 146.989,Z 735.187,A -85,B 0,C 180,E1 -25074.144,E2 -25074.144} C_VEL
LIN {X 0,Y 142.254,Z 744.083,A -85,B 0,C 180,E1 -25077.918,E2 -25077.918} C_VEL
LIN {X 0,Y 137.995,Z 751.242,A -85,B 0,C 180,E1 -25081.892,E2 -25081.892} C_VEL
LIN {X 0,Y 134.786,Z 756.074,A -85,B 0,C 180,E1 -25085.343,E2 -25085.343} C_VEL
LIN {X 0,Y 131.773,Z 760.76,A -85,B 0,C 180,E1 -25089.713,E2 -25089.713} C_VEL
LIN {X 0,Y 129.392,Z 764.341,A -85,B 0,C 180,E1 -25094.239,E2 -25094.239} C_VEL
LIN {X 0,Y 128.239,Z 766.188,A -85,B 0,C 180,E1 -25097.334,E2 -25097.334} C_VEL
LIN {X 0,Y 127.415,Z 767.575,A -85,B 0,C 180,E1 -25100.472,E2 -25100.472} C_VEL
LIN {X 0,Y 126.889,Z 768.561,A -85,B 0,C 180,E1 -25103.637,E2 -25103.637} C_VEL
LIN {X 0,Y 126.586,Z 769.167,A -85,B 0,C 180,E1 -25106.814,E2 -25106.814} C_VEL
LIN {X 0,Y 126.505,Z 769.393,A -85,B 0,C 180,E1 -25109.997,E2 -25109.997} C_VEL
LIN {X 0,Y 126.585,Z 769.198,A -85,B 0,C 180,E1 -25113.18,E2 -25113.18} C_VEL
LIN {X 0,Y 126.888,Z 768.613,A -85,B 0,C 180,E1 -25116.357,E2 -25116.357} C_VEL
LIN {X 0,Y 128.234,Z 766.293,A -85,B 0,C 180,E1 -25122.66,E2 -25122.66} C_VEL
LIN {X 0,Y 130.088,Z 763.421,A -85,B 0,C 180,E1 -25127.283,E2 -25127.283} C_VEL
LIN {X 0,Y 132.685,Z 759.524,A -85,B 0,C 180,E1 -25131.76,E2 -25131.76} C_VEL
LIN {X 0,Y 135.929,Z 754.503,A -85,B 0,C 180,E1 -25136.068,E2 -25136.068} C_VEL
LIN {X 0,Y 139.981,Z 748.169,A -85,B 0,C 180,E1 -25140.134,E2 -25140.134} C_VEL
LIN {X 0,Y 144.487,Z 740.234,A -85,B 0,C 180,E1 -25144.017,E2 -25144.017} C_VEL
LIN {X 0,Y 149.538,Z 730.395,A -85,B 0,C 180,E1 -25147.657,E2 -25147.657} C_VEL
LIN {X 0,Y 154.215,Z 720.038,A -85,B 0,C 180,E1 -25150.494,E2 -25150.494} C_VEL
LIN {X 0,Y 158.781,Z 708.359,A -85,B 0,C 180,E1 -25152.882,E2 -25152.882} C_VEL
LIN {X 0,Y 162.457,Z 696.684,A -85,B 0,C 180,E1 -25154.664,E2 -25154.664} C_VEL
LIN {X 0,Y 165.39,Z 684.533,A -85,B 0,C 180,E1 -25156.029,E2 -25156.029} C_VEL
LIN {X 0,Y 167.69,Z 671.519,A -85,B 0,C 180,E1 -25157.029,E2 -25157.029} C_VEL
LIN {X 0,Y 169.028,Z 658.087,A -85,B 0,C 180,E1 -25157.668,E2 -25157.668} C_VEL
LIN {X 0,Y 171.059,Z 629.38,A -85,B 0,C 180,E1 -25158.686,E2 -25158.686} C_VEL
LIN {X 0,Y 168.713,Z 623.775,A -85,B 0,C 180,E1 -25159.97,E2 -25159.97} C_VEL
LIN {X 0,Y 164.168,Z 615.311,A -85,B 0,C 180,E1 -25162.504,E2 -25162.504} C_VEL
LIN {X 0,Y 158.892,Z 606.429,A -85,B 0,C 180,E1 -25165.773,E2 -25165.773} C_VEL
LIN {X 0,Y 154.218,Z 599.339,A -85,B 0,C 180,E1 -25169.062,E2 -25169.062} C_VEL
LIN {X 0,Y 150.737,Z 594.609,A -85,B 0,C 180,E1 -25171.831,E2 -25171.831} C_VEL
LIN {X 0,Y 147.894,Z 590.678,A -85,B 0,C 180,E1 -25174.411,E2 -25174.411} C_VEL
LIN {X 0,Y 145.011,Z 587.17,A -85,B 0,C 180,E1 -25177.369,E2 -25177.369} C_VEL
LIN {X 0,Y 144.074,Z 585.664,A -85,B 0,C 180,E1 -25178.489,E2 -25178.489} C_VEL
LIN {X 0,Y 141.504,Z 583.19,A -85,B 0,C 180,E1 -25181.728,E2 -25181.728} C_VEL
LIN {X 0,Y 140.161,Z 580.434,A -85,B 0,C 180,E1 -25183.991,E2 -25183.991} C_VEL
LIN {X 0,Y 137.528,Z 578.608,A -85,B 0,C 180,E1 -25188.973,E2 -25188.973} C_VEL
LIN {X 0,Y 135.769,Z 574.803,A -85,B 0,C 180,E1 -25196.476,E2 -25196.476} C_VEL
LIN {X 0,Y 135.742,Z 574.452,A -85,B 0,C 180,E1 -25197.032,E2 -25197.032} C_VEL
LIN {X 0,Y 135.645,Z 574.403,A -85,B 0,C 180,E1 -25201.484,E2 -25201.484} C_VEL
LIN {X 0,Y 135.789,Z 574.846,A -85,B 0,C 180,E1 -25203.338,E2 -25203.338} C_VEL
LIN {X 0,Y 137.198,Z 578.192,A -85,B 0,C 180,E1 -25209.8,E2 -25209.8} C_VEL
LIN {X 0,Y 140.242,Z 580.7,A -85,B 0,C 180,E1 -25215.812,E2 -25215.812} C_VEL
LIN {X 0,Y 142.1,Z 583.972,A -85,B 0,C 180,E1 -25218.752,E2 -25218.752} C_VEL
LIN {X 0,Y 144.52,Z 586.24,A -85,B 0,C 180,E1 -25221.674,E2 -25221.674} C_VEL
LIN {X 0,Y 146.81,Z 589.613,A -85,B 0,C 180,E1 -25224.198,E2 -25224.198} C_VEL
LIN {X 0,Y 148.426,Z 591.354,A -85,B 0,C 180,E1 -25225.73,E2 -25225.73} C_VEL
LIN {X 0,Y 151.998,Z 596.331,A -85,B 0,C 180,E1 -25228.855,E2 -25228.855} C_VEL
LIN {X 0,Y 155.116,Z 600.781,A -85,B 0,C 180,E1 -25231.256,E2 -25231.256} C_VEL
LIN {X 0,Y 159.57,Z 608.997,A -85,B 0,C 180,E1 -25234.425,E2 -25234.425} C_VEL
LIN {X 0,Y 164.005,Z 618.289,A -85,B 0,C 180,E1 -25237.271,E2 -25237.271} C_VEL
LIN {X 0,Y 167.644,Z 627.087,A -85,B 0,C 180,E1 -25239.448,E2 -25239.448} C_VEL
LIN {X 0,Y 170.677,Z 635.844,A -85,B 0,C 180,E1 -25241.211,E2 -25241.211} C_VEL
LIN {X 0,Y 167.803,Z 673.309,A -85,B 0,C 180,E1 -25242.576,E2 -25242.576} C_VEL
LIN {X 0,Y 165.73,Z 686.862,A -85,B 0,C 180,E1 -25243.452,E2 -25243.452} C_VEL
LIN {X 0,Y 162.876,Z 699.124,A -85,B 0,C 180,E1 -25244.609,E2 -25244.609} C_VEL
LIN {X 0,Y 159.517,Z 710.201,A -85,B 0,C 180,E1 -25246.063,E2 -25246.063} C_VEL
LIN {X 0,Y 155.254,Z 721.75,A -85,B 0,C 180,E1 -25248.114,E2 -25248.114} C_VEL
LIN {X 0,Y 150.761,Z 732.153,A -85,B 0,C 180,E1 -25250.572,E2 -25250.572} C_VEL
LIN {X 0,Y 146.585,Z 740.664,A -85,B 0,C 180,E1 -25253.183,E2 -25253.183} C_VEL
LIN {X 0,Y 142.344,Z 748.516,A -85,B 0,C 180,E1 -25256.262,E2 -25256.262} C_VEL
LIN {X 0,Y 138.051,Z 756.043,A -85,B 0,C 180,E1 -25260.131,E2 -25260.131} C_VEL
LIN {X 0,Y 134.714,Z 761.455,A -85,B 0,C 180,E1 -25263.68,E2 -25263.68} C_VEL
LIN {X 0,Y 131.495,Z 766.555,A -85,B 0,C 180,E1 -25268.033,E2 -25268.033} C_VEL
LIN {X 0,Y 129.05,Z 770.524,A -85,B 0,C 180,E1 -25272.574,E2 -25272.574} C_VEL
LIN {X 0,Y 127.451,Z 773.485,A -85,B 0,C 180,E1 -25277.312,E2 -25277.312} C_VEL
LIN {X 0,Y 126.792,Z 774.861,A -85,B 0,C 180,E1 -25280.431,E2 -25280.431} C_VEL
LIN {X 0,Y 126.411,Z 775.86,A -85,B 0,C 180,E1 -25283.619,E2 -25283.619} C_VEL
LIN {X 0,Y 126.303,Z 776.471,A -85,B 0,C 180,E1 -25286.813,E2 -25286.813} C_VEL
LIN {X 0,Y 126.427,Z 776.612,A -85,B 0,C 180,E1 -25291.049,E2 -25291.049} C_VEL
LIN {X 0,Y 125.904,Z 776.378,A -85,B 0,C 180,E1 -25293.718,E2 -25293.718} C_VEL
LIN {X 0,Y 123.718,Z 775.317,A -85,B 0,C 180,E1 -25298.138,E2 -25298.138} C_VEL
LIN {X 0,Y 122.335,Z 773.946,A -85,B 0,C 180,E1 -25301.741,E2 -25301.741} C_VEL
LIN {X 0,Y 122.421,Z 772.626,A -85,B 0,C 180,E1 -25304.446,E2 -25304.446} C_VEL
LIN {X 0,Y 122.781,Z 772.087,A -85,B 0,C 180,E1 -25305.325,E2 -25305.325} C_VEL
LIN {X 0,Y 126.785,Z 768.256,A -85,B 0,C 180,E1 -25310.909,E2 -25310.909} C_VEL
LIN {X 0,Y 130.973,Z 774.006,A -85,B 0,C 180,E1 -25317.139,E2 -25317.139} C_VEL
LIN {X 0,Y 135.308,Z 777.272,A -85,B 0,C 180,E1 -25321.295,E2 -25321.295} C_VEL
LIN {X 0,Y 138.929,Z 779.039,A -85,B 0,C 180,E1 -25323.814,E2 -25323.814} C_VEL
LIN {X 0,Y 142.837,Z 780.342,A -85,B 0,C 180,E1 -25326.191,E2 -25326.191} C_VEL
LIN {X 0,Y 151.81,Z 781.863,A -85,B 0,C 180,E1 -25330.403,E2 -25330.403} C_VEL
LIN {X 0,Y 156.789,Z 782.084,A -85,B 0,C 180,E1 -25332.253,E2 -25332.253} C_VEL
LIN {X 0,Y 167.475,Z 781.211,A -85,B 0,C 180,E1 -25335.514,E2 -25335.514} C_VEL
LIN {X 0,Y 167.906,Z 781.127,A -85,B 0,C 180,E1 -25336.241,E2 -25336.241} C_VEL
LIN {X 0,Y 159.622,Z 781.823,A -85,B 0,C 180,E1 -25338.667,E2 -25338.667} C_VEL
LIN {X 0,Y 149.638,Z 781.203,A -85,B 0,C 180,E1 -25342.369,E2 -25342.369} C_VEL
LIN {X 0,Y 145.077,Z 780.281,A -85,B 0,C 180,E1 -25344.457,E2 -25344.457} C_VEL
LIN {X 0,Y 137.145,Z 777.103,A -85,B 0,C 180,E1 -25349.173,E2 -25349.173} C_VEL
LIN {X 0,Y 132.348,Z 773.675,A -85,B 0,C 180,E1 -25353.168,E2 -25353.168} C_VEL
LIN {X 0,Y 128.702,Z 769.348,A -85,B 0,C 180,E1 -25357.527,E2 -25357.527} C_VEL
LIN {X 0,Y 126.072,Z 763.395,A -85,B 0,C 180,E1 -25362.601,E2 -25362.601} C_VEL
LIN {X 0,Y 124.836,Z 755.978,A -85,B 0,C 180,E1 -25367.812,E2 -25367.812} C_VEL
LIN {X 0,Y 124.879,Z 747.38,A -85,B 0,C 180,E1 -25372.725,E2 -25372.725} C_VEL
LIN {X 0,Y 125.242,Z 740.18,A -85,B 0,C 180,E1 -25375.978,E2 -25375.978} C_VEL
LIN {X 0,Y 125.386,Z 732.029,A -85,B 0,C 180,E1 -25378.796,E2 -25378.796} C_VEL
LIN {X 0,Y 125.49,Z 723.186,A -85,B 0,C 180,E1 -25381.204,E2 -25381.204} C_VEL
LIN {X 0,Y 125.652,Z 711.548,A -85,B 0,C 180,E1 -25383.608,E2 -25383.608} C_VEL
LIN {X 0,Y 125.641,Z 698.268,A -85,B 0,C 180,E1 -25385.517,E2 -25385.517} C_VEL
LIN {X 0,Y 125.231,Z 675.893,A -85,B 0,C 180,E1 -25388.37,E2 -25388.37} C_VEL
LIN {X 0,Y 124.883,Z 672.573,A -85,B 0,C 180,E1 -25389.311,E2 -25389.311} C_VEL
LIN {X 0,Y 124.839,Z 671.562,A -85,B 0,C 180,E1 -25390.133,E2 -25390.133} C_VEL
LIN {X 0,Y 125.072,Z 671.397,A -85,B 0,C 180,E1 -25390.728,E2 -25390.728} C_VEL
LIN {X 0,Y 125.775,Z 669.832,A -85,B 0,C 180,E1 -25391.687,E2 -25391.687} C_VEL
LIN {X 0,Y 127.044,Z 665.785,A -85,B 0,C 180,E1 -25392.881,E2 -25392.881} C_VEL
LIN {X 0,Y 129.396,Z 655.41,A -85,B 0,C 180,E1 -25394.666,E2 -25394.666} C_VEL
LIN {X 0,Y 130.483,Z 650.701,A -85,B 0,C 180,E1 -25395.479,E2 -25395.479} C_VEL
LIN {X 0,Y 131.612,Z 649.033,A -85,B 0,C 180,E1 -25396.88,E2 -25396.88} C_VEL
LIN {X 0,Y 132.884,Z 645.961,A -85,B 0,C 180,E1 -25398.103,E2 -25398.103} C_VEL
LIN {X 0,Y 134.73,Z 640.071,A -85,B 0,C 180,E1 -25399.483,E2 -25399.483} C_VEL
LIN {X 0,Y 136.596,Z 636.568,A -85,B 0,C 180,E1 -25401.11,E2 -25401.11} C_VEL
LIN {X 0,Y 138.508,Z 635.712,A -85,B 0,C 180,E1 -25402.982,E2 -25402.982} C_VEL
LIN {X 0,Y 141.439,Z 632.836,A -85,B 0,C 180,E1 -25405.328,E2 -25405.328} C_VEL
LIN {X 0,Y 145.616,Z 627.342,A -85,B 0,C 180,E1 -25408.072,E2 -25408.072} C_VEL
LIN {X 0,Y 146.596,Z 625.938,A -85,B 0,C 180,E1 -25408.647,E2 -25408.647} C_VEL
LIN {X 0,Y 149.792,Z 624.428,A -85,B 0,C 180,E1 -25410.69,E2 -25410.69} C_VEL
LIN {X 0,Y 153.669,Z 621.274,A -85,B 0,C 180,E1 -25412.798,E2 -25412.798} C_VEL
LIN {X 0,Y 156.226,Z 618.615,A -85,B 0,C 180,E1 -25414.023,E2 -25414.023} C_VEL
LIN {X 0,Y 159.052,Z 617.741,A -85,B 0,C 180,E1 -25415.448,E2 -25415.448} C_VEL
LIN {X 0,Y 161.376,Z 621.609,A -85,B 0,C 180,E1 -25416.883,E2 -25416.883} C_VEL
LIN {X 0,Y 165.669,Z 630.315,A -85,B 0,C 180,E1 -25419.423,E2 -25419.423} C_VEL
LIN {X 0,Y 166.112,Z 631.455,A -85,B 0,C 180,E1 -25419.686,E2 -25419.686} C_VEL
LIN {X 0,Y 163.388,Z 666.598,A -85,B 0,C 180,E1 -25421.004,E2 -25421.004} C_VEL
LIN {X 0,Y 161.332,Z 679.891,A -85,B 0,C 180,E1 -25421.863,E2 -25421.863} C_VEL
LIN {X 0,Y 158.707,Z 691.857,A -85,B 0,C 180,E1 -25423.055,E2 -25423.055} C_VEL
LIN {X 0,Y 155.404,Z 703.124,A -85,B 0,C 180,E1 -25424.576,E2 -25424.576} C_VEL
LIN {X 0,Y 151.065,Z 714.745,A -85,B 0,C 180,E1 -25426.666,E2 -25426.666} C_VEL
LIN {X 0,Y 146.461,Z 725.185,A -85,B 0,C 180,E1 -25429.168,E2 -25429.168} C_VEL
LIN {X 0,Y 142.209,Z 733.709,A -85,B 0,C 180,E1 -25431.845,E2 -25431.845} C_VEL
LIN {X 0,Y 137.872,Z 741.563,A -85,B 0,C 180,E1 -25435.006,E2 -25435.006} C_VEL
LIN {X 0,Y 133.198,Z 749.23,A -85,B 0,C 180,E1 -25439.037,E2 -25439.037} C_VEL
LIN {X 0,Y 128.358,Z 756.281,A -85,B 0,C 180,E1 -25444.019,E2 -25444.019} C_VEL
LIN {X 0,Y 125.131,Z 760.966,A -85,B 0,C 180,E1 -25448.585,E2 -25448.585} C_VEL
LIN {X 0,Y 122.575,Z 764.547,A -85,B 0,C 180,E1 -25453.338,E2 -25453.338} C_VEL
LIN {X 0,Y 121.331,Z 766.393,A -85,B 0,C 180,E1 -25456.6,E2 -25456.6} C_VEL
LIN {X 0,Y 120.43,Z 767.78,A -85,B 0,C 180,E1 -25459.914,E2 -25459.914} C_VEL
LIN {X 0,Y 119.841,Z 768.766,A -85,B 0,C 180,E1 -25463.261,E2 -25463.261} C_VEL
LIN {X 0,Y 119.499,Z 769.372,A -85,B 0,C 180,E1 -25466.625,E2 -25466.625} C_VEL
LIN {X 0,Y 119.419,Z 769.597,A -85,B 0,C 180,E1 -25469.997,E2 -25469.997} C_VEL
LIN {X 0,Y 119.498,Z 769.402,A -85,B 0,C 180,E1 -25473.369,E2 -25473.369} C_VEL
LIN {X 0,Y 119.84,Z 768.817,A -85,B 0,C 180,E1 -25476.733,E2 -25476.733} C_VEL
LIN {X 0,Y 121.327,Z 766.497,A -85,B 0,C 180,E1 -25483.394,E2 -25483.394} C_VEL
LIN {X 0,Y 123.309,Z 763.626,A -85,B 0,C 180,E1 -25488.265,E2 -25488.265} C_VEL
LIN {X 0,Y 126.097,Z 759.729,A -85,B 0,C 180,E1 -25492.96,E2 -25492.96} C_VEL
LIN {X 0,Y 129.587,Z 754.706,A -85,B 0,C 180,E1 -25497.447,E2 -25497.447} C_VEL
LIN {X 0,Y 133.877,Z 748.372,A -85,B 0,C 180,E1 -25501.662,E2 -25501.662} C_VEL
LIN {X 0,Y 138.383,Z 740.922,A -85,B 0,C 180,E1 -25505.447,E2 -25505.447} C_VEL
LIN {X 0,Y 143.052,Z 732.375,A -85,B 0,C 180,E1 -25508.781,E2 -25508.781} C_VEL
LIN {X 0,Y 147.867,Z 722.514,A -85,B 0,C 180,E1 -25511.71,E2 -25511.71} C_VEL
LIN {X 0,Y 152.559,Z 711.404,A -85,B 0,C 180,E1 -25514.165,E2 -25514.165} C_VEL
LIN {X 0,Y 156.387,Z 700.506,A -85,B 0,C 180,E1 -25515.971,E2 -25515.971} C_VEL
LIN {X 0,Y 159.711,Z 688.448,A -85,B 0,C 180,E1 -25517.479,E2 -25517.479} C_VEL
LIN {X 0,Y 162.334,Z 675.572,A -85,B 0,C 180,E1 -25518.601,E2 -25518.601} C_VEL
LIN {X 0,Y 164.035,Z 662.058,A -85,B 0,C 180,E1 -25519.344,E2 -25519.344} C_VEL
LIN {X 0,Y 166.301,Z 631.682,A -85,B 0,C 180,E1 -25520.446,E2 -25520.446} C_VEL
LIN {X 0,Y 163.525,Z 625.637,A -85,B 0,C 180,E1 -25522.069,E2 -25522.069} C_VEL
LIN {X 0,Y 157.742,Z 615.08,A -85,B 0,C 180,E1 -25525.702,E2 -25525.702} C_VEL
LIN {X 0,Y 153.318,Z 607.9,A -85,B 0,C 180,E1 -25528.86,E2 -25528.86} C_VEL
LIN {X 0,Y 150.331,Z 603.472,A -85,B 0,C 180,E1 -25531.243,E2 -25531.243} C_VEL
LIN {X 0,Y 148.449,Z 600.742,A -85,B 0,C 180,E1 -25532.891,E2 -25532.891} C_VEL
LIN {X 0,Y 145.857,Z 597.021,A -85,B 0,C 180,E1 -25535.402,E2 -25535.402} C_VEL
LIN {X 0,Y 143.085,Z 593.45,A -85,B 0,C 180,E1 -25538.451,E2 -25538.451} C_VEL
LIN {X 0,Y 142.372,Z 592.313,A -85,B 0,C 180,E1 -25539.357,E2 -25539.357} C_VEL
LIN {X 0,Y 139.725,Z 589.385,A -85,B 0,C 180,E1 -25543,E2 -25543} C_VEL
LIN {X 0,Y 138.659,Z 587.234,A -85,B 0,C 180,E1 -25544.944,E2 -25544.944} C_VEL
LIN {X 0,Y 136.092,Z 585.079,A -85,B 0,C 180,E1 -25550.451,E2 -25550.451} C_VEL
LIN {X 0,Y 134.808,Z 581.462,A -85,B 0,C 180,E1 -25557.759,E2 -25557.759} C_VEL
LIN {X 0,Y 134.857,Z 581.657,A -85,B 0,C 180,E1 -25562.613,E2 -25562.613} C_VEL
LIN {X 0,Y 135.587,Z 584.172,A -85,B 0,C 180,E1 -25567.445,E2 -25567.445} C_VEL
LIN {X 0,Y 138.237,Z 587.002,A -85,B 0,C 180,E1 -25573.974,E2 -25573.974} C_VEL
LIN {X 0,Y 138.887,Z 587.645,A -85,B 0,C 180,E1 -25575.124,E2 -25575.124} C_VEL
LIN {X 0,Y 140.836,Z 590.89,A -85,B 0,C 180,E1 -25578.314,E2 -25578.314} C_VEL
LIN {X 0,Y 142.807,Z 592.913,A -85,B 0,C 180,E1 -25580.827,E2 -25580.827} C_VEL
LIN {X 0,Y 145.28,Z 596.446,A -85,B 0,C 180,E1 -25583.664,E2 -25583.664} C_VEL
LIN {X 0,Y 146.519,Z 597.978,A -85,B 0,C 180,E1 -25584.911,E2 -25584.911} C_VEL
LIN {X 0,Y 149.835,Z 602.733,A -85,B 0,C 180,E1 -25587.972,E2 -25587.972} C_VEL
LIN {X 0,Y 152.331,Z 606.414,A -85,B 0,C 180,E1 -25590.019,E2 -25590.019} C_VEL
LIN {X 0,Y 156.491,Z 614.482,A -85,B 0,C 180,E1 -25593.206,E2 -25593.206} C_VEL
LIN {X 0,Y 160.361,Z 622.962,A -85,B 0,C 180,E1 -25595.886,E2 -25595.886} C_VEL
LIN {X 0,Y 163.946,Z 632.093,A -85,B 0,C 180,E1 -25598.208,E2 -25598.208} C_VEL
LIN {X 0,Y 165.928,Z 637.798,A -85,B 0,C 180,E1 -25599.445,E2 -25599.445} C_VEL
LIN {X 0,Y 163.099,Z 672.954,A -85,B 0,C 180,E1 -25600.729,E2 -25600.729} C_VEL
LIN {X 0,Y 161.034,Z 686.273,A -85,B 0,C 180,E1 -25601.598,E2 -25601.598} C_VEL
LIN {X 0,Y 157.981,Z 698.926,A -85,B 0,C 180,E1 -25602.779,E2 -25602.779} C_VEL
LIN {X 0,Y 154.488,Z 710.002,A -85,B 0,C 180,E1 -25604.237,E2 -25604.237} C_VEL
LIN {X 0,Y 150.049,Z 721.549,A -85,B 0,C 180,E1 -25606.305,E2 -25606.305} C_VEL
LIN {X 0,Y 145.336,Z 731.951,A -85,B 0,C 180,E1 -25608.79,E2 -25608.79} C_VEL
LIN {X 0,Y 140.943,Z 740.461,A -85,B 0,C 180,E1 -25611.446,E2 -25611.446} C_VEL
LIN {X 0,Y 136.469,Z 748.312,A -85,B 0,C 180,E1 -25614.598,E2 -25614.598} C_VEL
LIN {X 0,Y 131.519,Z 756.435,A -85,B 0,C 180,E1 -25618.959,E2 -25618.959} C_VEL
LIN {X 0,Y 127.11,Z 763.071,A -85,B 0,C 180,E1 -25623.751,E2 -25623.751} C_VEL
LIN {X 0,Y 123.932,Z 767.785,A -85,B 0,C 180,E1 -25628.374,E2 -25628.374} C_VEL
LIN {X 0,Y 121.605,Z 771.396,A -85,B 0,C 180,E1 -25633.207,E2 -25633.207} C_VEL
LIN {X 0,Y 120.524,Z 773.259,A -85,B 0,C 180,E1 -25636.515,E2 -25636.515} C_VEL
LIN {X 0,Y 119.784,Z 774.656,A -85,B 0,C 180,E1 -25639.865,E2 -25639.865} C_VEL
LIN {X 0,Y 119.219,Z 776.267,A -85,B 0,C 180,E1 -25646.623,E2 -25646.623} C_VEL
LIN {X 0,Y 119.338,Z 776.41,A -85,B 0,C 180,E1 -25651.083,E2 -25651.083} C_VEL
LIN {X 0,Y 119.92,Z 775.642,A -85,B 0,C 180,E1 -25656.734,E2 -25656.734} C_VEL
LIN {X 0,Y 120.698,Z 774.64,A -85,B 0,C 180,E1 -25660.063,E2 -25660.063} C_VEL
LIN {X 0,Y 122.781,Z 772.087,A -85,B 0,C 180,E1 -25665.325,E2 -25665.325} C_VEL
LIN {X 0,Y 123.197,Z 771.009,A -85,B 0,C 180,E1 -25667.161,E2 -25667.161} C_VEL
LIN {X 0,Y 122.514,Z 768.913,A -85,B 0,C 180,E1 -25670.252,E2 -25670.252} C_VEL
LIN {X 0,Y 121.957,Z 767.775,A -85,B 0,C 180,E1 -25673.048,E2 -25673.048} C_VEL
LIN {X 0,Y 122.2,Z 768.073,A -85,B 0,C 180,E1 -25674.574,E2 -25674.574} C_VEL
LIN {X 0,Y 122.48,Z 768.502,A -85,B 0,C 180,E1 -25675.136,E2 -25675.136} C_VEL
LIN {X 0,Y 126.364,Z 773.114,A -85,B 0,C 180,E1 -25680.04,E2 -25680.04} C_VEL
LIN {X 0,Y 131.331,Z 776.517,A -85,B 0,C 180,E1 -25684.19,E2 -25684.19} C_VEL
LIN {X 0,Y 137.259,Z 779.106,A -85,B 0,C 180,E1 -25687.914,E2 -25687.914} C_VEL
LIN {X 0,Y 141.71,Z 780.384,A -85,B 0,C 180,E1 -25690.148,E2 -25690.148} C_VEL
LIN {X 0,Y 151.603,Z 781.786,A -85,B 0,C 180,E1 -25694.059,E2 -25694.059} C_VEL
LIN {X 0,Y 157.007,Z 781.986,A -85,B 0,C 180,E1 -25695.744,E2 -25695.744} C_VEL
LIN {X 0,Y 154.342,Z 781.839,A -85,B 0,C 180,E1 -25696.919,E2 -25696.919} C_VEL
LIN {X 0,Y 149.114,Z 781.43,A -85,B 0,C 180,E1 -25698.712,E2 -25698.712} C_VEL
LIN {X 0,Y 144.099,Z 780.524,A -85,B 0,C 180,E1 -25700.651,E2 -25700.651} C_VEL
LIN {X 0,Y 139.429,Z 779.203,A -85,B 0,C 180,E1 -25702.781,E2 -25702.781} C_VEL
LIN {X 0,Y 133.163,Z 776.541,A -85,B 0,C 180,E1 -25706.347,E2 -25706.347} C_VEL
LIN {X 0,Y 127.831,Z 772.984,A -85,B 0,C 180,E1 -25710.343,E2 -25710.343} C_VEL
LIN {X 0,Y 123.724,Z 768.521,A -85,B 0,C 180,E1 -25714.784,E2 -25714.784} C_VEL
LIN {X 0,Y 120.487,Z 762.064,A -85,B 0,C 180,E1 -25720.315,E2 -25720.315} C_VEL
LIN {X 0,Y 118.981,Z 754.94,A -85,B 0,C 180,E1 -25725.461,E2 -25725.461} C_VEL
LIN {X 0,Y 118.767,Z 746.446,A -85,B 0,C 180,E1 -25730.635,E2 -25730.635} C_VEL
LIN {X 0,Y 119.146,Z 738.204,A -85,B 0,C 180,E1 -25734.5,E2 -25734.5} C_VEL
LIN {X 0,Y 119.237,Z 729.96,A -85,B 0,C 180,E1 -25737.467,E2 -25737.467} C_VEL
LIN {X 0,Y 119.215,Z 720.96,A -85,B 0,C 180,E1 -25740,E2 -25740} C_VEL
LIN {X 0,Y 119.332,Z 710.33,A -85,B 0,C 180,E1 -25742.215,E2 -25742.215} C_VEL
LIN {X 0,Y 119.056,Z 692.934,A -85,B 0,C 180,E1 -25744.868,E2 -25744.868} C_VEL
LIN {X 0,Y 118.529,Z 690.644,A -85,B 0,C 180,E1 -25745.849,E2 -25745.849} C_VEL
LIN {X 0,Y 118.405,Z 690.383,A -85,B 0,C 180,E1 -25746.39,E2 -25746.39} C_VEL
LIN {X 0,Y 118.424,Z 690.465,A -85,B 0,C 180,E1 -25746.817,E2 -25746.817} C_VEL
LIN {X 0,Y 119.392,Z 688.999,A -85,B 0,C 180,E1 -25748.464,E2 -25748.464} C_VEL
LIN {X 0,Y 120.834,Z 685.874,A -85,B 0,C 180,E1 -25749.669,E2 -25749.669} C_VEL
LIN {X 0,Y 123.719,Z 678.372,A -85,B 0,C 180,E1 -25751.364,E2 -25751.364} C_VEL
LIN {X 0,Y 124.794,Z 676.856,A -85,B 0,C 180,E1 -25752.915,E2 -25752.915} C_VEL
LIN {X 0,Y 126.43,Z 673.451,A -85,B 0,C 180,E1 -25754.486,E2 -25754.486} C_VEL
LIN {X 0,Y 128.225,Z 668.428,A -85,B 0,C 180,E1 -25755.804,E2 -25755.804} C_VEL
LIN {X 0,Y 130.87,Z 658.087,A -85,B 0,C 180,E1 -25757.482,E2 -25757.482} C_VEL
LIN {X 0,Y 131.362,Z 656.129,A -85,B 0,C 180,E1 -25757.816,E2 -25757.816} C_VEL
LIN {X 0,Y 133.114,Z 652.903,A -85,B 0,C 180,E1 -25759.548,E2 -25759.548} C_VEL
LIN {X 0,Y 134.832,Z 648.56,A -85,B 0,C 180,E1 -25760.899,E2 -25760.899} C_VEL
LIN {X 0,Y 136.223,Z 644.52,A -85,B 0,C 180,E1 -25761.838,E2 -25761.838} C_VEL
LIN {X 0,Y 136.97,Z 643.327,A -85,B 0,C 180,E1 -25762.453,E2 -25762.453} C_VEL
LIN {X 0,Y 139.387,Z 641.778,A -85,B 0,C 180,E1 -25764.581,E2 -25764.581} C_VEL
LIN {X 0,Y 142.687,Z 638.514,A -85,B 0,C 180,E1 -25767.005,E2 -25767.005} C_VEL
LIN {X 0,Y 147.443,Z 632.549,A -85,B 0,C 180,E1 -25769.893,E2 -25769.893} C_VEL
LIN {X 0,Y 151.693,Z 630.145,A -85,B 0,C 180,E1 -25772.391,E2 -25772.391} C_VEL
LIN {X 0,Y 156.336,Z 626.04,A -85,B 0,C 180,E1 -25774.678,E2 -25774.678} C_VEL
LIN {X 0,Y 157.277,Z 625.375,A -85,B 0,C 180,E1 -25775.123,E2 -25775.123} C_VEL
LIN {X 0,Y 161.52,Z 634.013,A -85,B 0,C 180,E1 -25777.846,E2 -25777.846} C_VEL
LIN {X 0,Y 158.812,Z 666.969,A -85,B 0,C 180,E1 -25779.084,E2 -25779.084} C_VEL
LIN {X 0,Y 156.737,Z 679.875,A -85,B 0,C 180,E1 -25779.915,E2 -25779.915} C_VEL
LIN {X 0,Y 153.962,Z 692.068,A -85,B 0,C 180,E1 -25781.13,E2 -25781.13} C_VEL
LIN {X 0,Y 150.522,Z 703.333,A -85,B 0,C 180,E1 -25782.657,E2 -25782.657} C_VEL
LIN {X 0,Y 145.996,Z 714.953,A -85,B 0,C 180,E1 -25784.759,E2 -25784.759} C_VEL
LIN {X 0,Y 141.16,Z 725.393,A -85,B 0,C 180,E1 -25787.282,E2 -25787.282} C_VEL
LIN {X 0,Y 136.687,Z 733.917,A -85,B 0,C 180,E1 -25790.003,E2 -25790.003} C_VEL
LIN {X 0,Y 131.974,Z 742.009,A -85,B 0,C 180,E1 -25793.348,E2 -25793.348} C_VEL
LIN {X 0,Y 127.164,Z 749.436,A -85,B 0,C 180,E1 -25797.391,E2 -25797.391} C_VEL
LIN {X 0,Y 122.011,Z 756.487,A -85,B 0,C 180,E1 -25802.557,E2 -25802.557} C_VEL
LIN {X 0,Y 118.549,Z 761.172,A -85,B 0,C 180,E1 -25807.332,E2 -25807.332} C_VEL
LIN {X 0,Y 115.796,Z 764.752,A -85,B 0,C 180,E1 -25812.331,E2 -25812.331} C_VEL
LIN {X 0,Y 114.429,Z 766.599,A -85,B 0,C 180,E1 -25815.775,E2 -25815.775} C_VEL
LIN {X 0,Y 113.434,Z 767.985,A -85,B 0,C 180,E1 -25819.285,E2 -25819.285} C_VEL
LIN {X 0,Y 112.791,Z 768.971,A -85,B 0,C 180,E1 -25822.838,E2 -25822.838} C_VEL
LIN {X 0,Y 112.425,Z 769.576,A -85,B 0,C 180,E1 -25826.413,E2 -25826.413} C_VEL
LIN {X 0,Y 112.335,Z 769.801,A -85,B 0,C 180,E1 -25829.997,E2 -25829.997} C_VEL
LIN {X 0,Y 112.424,Z 769.606,A -85,B 0,C 180,E1 -25833.581,E2 -25833.581} C_VEL
LIN {X 0,Y 112.789,Z 769.022,A -85,B 0,C 180,E1 -25837.156,E2 -25837.156} C_VEL
LIN {X 0,Y 114.424,Z 766.701,A -85,B 0,C 180,E1 -25844.219,E2 -25844.219} C_VEL
LIN {X 0,Y 116.577,Z 763.83,A -85,B 0,C 180,E1 -25849.361,E2 -25849.361} C_VEL
LIN {X 0,Y 119.57,Z 759.933,A -85,B 0,C 180,E1 -25854.292,E2 -25854.292} C_VEL
LIN {X 0,Y 123.332,Z 754.909,A -85,B 0,C 180,E1 -25858.967,E2 -25858.967} C_VEL
LIN {X 0,Y 127.881,Z 748.575,A -85,B 0,C 180,E1 -25863.334,E2 -25863.334} C_VEL
LIN {X 0,Y 132.359,Z 741.627,A -85,B 0,C 180,E1 -25867.001,E2 -25867.001} C_VEL
LIN {X 0,Y 137.579,Z 732.577,A -85,B 0,C 180,E1 -25870.637,E2 -25870.637} C_VEL
LIN {X 0,Y 142.643,Z 722.715,A -85,B 0,C 180,E1 -25873.609,E2 -25873.609} C_VEL
LIN {X 0,Y 147.563,Z 711.603,A -85,B 0,C 180,E1 -25876.08,E2 -25876.08} C_VEL
LIN {X 0,Y 151.543,Z 700.704,A -85,B 0,C 180,E1 -25877.9,E2 -25877.9} C_VEL
LIN {X 0,Y 155.008,Z 688.645,A -85,B 0,C 180,E1 -25879.41,E2 -25879.41} C_VEL
LIN {X 0,Y 157.685,Z 676.08,A -85,B 0,C 180,E1 -25880.512,E2 -25880.512} C_VEL
LIN {X 0,Y 159.433,Z 663.183,A -85,B 0,C 180,E1 -25881.23,E2 -25881.23} C_VEL
LIN {X 0,Y 161.697,Z 634.125,A -85,B 0,C 180,E1 -25882.303,E2 -25882.303} C_VEL
LIN {X 0,Y 156.561,Z 623.943,A -85,B 0,C 180,E1 -25885.63,E2 -25885.63} C_VEL
LIN {X 0,Y 151.464,Z 614.881,A -85,B 0,C 180,E1 -25889.403,E2 -25889.403} C_VEL
LIN {X 0,Y 146.639,Z 607.395,A -85,B 0,C 180,E1 -25893.588,E2 -25893.588} C_VEL
LIN {X 0,Y 143.836,Z 603.374,A -85,B 0,C 180,E1 -25896.443,E2 -25896.443} C_VEL
LIN {X 0,Y 141.059,Z 599.405,A -85,B 0,C 180,E1 -25899.778,E2 -25899.778} C_VEL
LIN {X 0,Y 138.019,Z 595.559,A -85,B 0,C 180,E1 -25904.305,E2 -25904.305} C_VEL
LIN {X 0,Y 137.298,Z 594.069,A -85,B 0,C 180,E1 -25905.739,E2 -25905.739} C_VEL
LIN {X 0,Y 134.66,Z 591.351,A -85,B 0,C 180,E1 -25912.314,E2 -25912.314} C_VEL
LIN {X 0,Y 133.931,Z 588.609,A -85,B 0,C 180,E1 -25917.744,E2 -25917.744} C_VEL
LIN {X 0,Y 133.936,Z 588.558,A -85,B 0,C 180,E1 -25921.879,E2 -25921.879} C_VEL
LIN {X 0,Y 135.913,Z 593.041,A -85,B 0,C 180,E1 -25931.076,E2 -25931.076} C_VEL
LIN {X 0,Y 137.473,Z 594.333,A -85,B 0,C 180,E1 -25934.243,E2 -25934.243} C_VEL
LIN {X 0,Y 139.516,Z 597.783,A -85,B 0,C 180,E1 -25937.782,E2 -25937.782} C_VEL
LIN {X 0,Y 141.105,Z 599.522,A -85,B 0,C 180,E1 -25939.93,E2 -25939.93} C_VEL
LIN {X 0,Y 143.817,Z 603.329,A -85,B 0,C 180,E1 -25943.173,E2 -25943.173} C_VEL
LIN {X 0,Y 147.453,Z 608.737,A -85,B 0,C 180,E1 -25946.828,E2 -25946.828} C_VEL
LIN {X 0,Y 150.065,Z 612.834,A -85,B 0,C 180,E1 -25949.119,E2 -25949.119} C_VEL
LIN {X 0,Y 154.301,Z 621.675,A -85,B 0,C 180,E1 -25952.563,E2 -25952.563} C_VEL
LIN {X 0,Y 158.557,Z 632.008,A -85,B 0,C 180,E1 -25955.672,E2 -25955.672} C_VEL
LIN {X 0,Y 161.31,Z 640.128,A -85,B 0,C 180,E1 -25957.586,E2 -25957.586} C_VEL
LIN {X 0,Y 158.579,Z 672.678,A -85,B 0,C 180,E1 -25958.784,E2 -25958.784} C_VEL
LIN {X 0,Y 156.342,Z 686.421,A -85,B 0,C 180,E1 -25959.679,E2 -25959.679} C_VEL
LIN {X 0,Y 153.258,Z 698.728,A -85,B 0,C 180,E1 -25960.835,E2 -25960.835} C_VEL
LIN {X 0,Y 149.625,Z 709.802,A -85,B 0,C 180,E1 -25962.291,E2 -25962.291} C_VEL
LIN {X 0,Y 144.988,Z 721.348,A -85,B 0,C 180,E1 -25964.363,E2 -25964.363} C_VEL
LIN {X 0,Y 140.074,Z 731.75,A -85,B 0,C 180,E1 -25966.877,E2 -25966.877} C_VEL
LIN {X 0,Y 135.434,Z 740.258,A -85,B 0,C 180,E1 -25969.564,E2 -25969.564} C_VEL
LIN {X 0,Y 129.834,Z 749.482,A -85,B 0,C 180,E1 -25973.46,E2 -25973.46} C_VEL
LIN {X 0,Y 125.048,Z 756.827,A -85,B 0,C 180,E1 -25977.665,E2 -25977.665} C_VEL
LIN {X 0,Y 120.759,Z 762.867,A -85,B 0,C 180,E1 -25982.255,E2 -25982.255} C_VEL
LIN {X 0,Y 117.346,Z 767.581,A -85,B 0,C 180,E1 -25987.093,E2 -25987.093} C_VEL
LIN {X 0,Y 114.774,Z 771.19,A -85,B 0,C 180,E1 -25992.175,E2 -25992.175} C_VEL
LIN {X 0,Y 113.615,Z 773.054,A -85,B 0,C 180,E1 -25995.678,E2 -25995.678} C_VEL
LIN {X 0,Y 112.776,Z 774.451,A -85,B 0,C 180,E1 -25999.228,E2 -25999.228} C_VEL
LIN {X 0,Y 112.126,Z 776.062,A -85,B 0,C 180,E1 -26006.41,E2 -26006.41} C_VEL
LIN {X 0,Y 112.25,Z 776.277,A -85,B 0,C 180,E1 -26010.003,E2 -26010.003} C_VEL
LIN {X 0,Y 112.42,Z 776.052,A -85,B 0,C 180,E1 -26013.587,E2 -26013.587} C_VEL
LIN {X 0,Y 113.716,Z 774.435,A -85,B 0,C 180,E1 -26020.688,E2 -26020.688} C_VEL
LIN {X 0,Y 115.901,Z 771.938,A -85,B 0,C 180,E1 -26026.15,E2 -26026.15} C_VEL
LIN {X 0,Y 119.035,Z 768.887,A -85,B 0,C 180,E1 -26030.75,E2 -26030.75} C_VEL
LIN {X 0,Y 121.392,Z 766.833,A -85,B 0,C 180,E1 -26033.345,E2 -26033.345} C_VEL
LIN {X 0,Y 122.48,Z 768.502,A -85,B 0,C 180,E1 -26035.136,E2 -26035.136} C_VEL
LIN {X 0,Y 122.995,Z 769.856,A -85,B 0,C 180,E1 -26036.878,E2 -26036.878} C_VEL
LIN {X 0,Y 122.815,Z 772.387,A -85,B 0,C 180,E1 -26043.075,E2 -26043.075} C_VEL
LIN {X 0,Y 124.14,Z 773.441,A -85,B 0,C 180,E1 -26044.742,E2 -26044.742} C_VEL
LIN {X 0,Y 127.714,Z 775.633,A -85,B 0,C 180,E1 -26047.255,E2 -26047.255} C_VEL
LIN {X 0,Y 136.459,Z 779.111,A -85,B 0,C 180,E1 -26052.034,E2 -26052.034} C_VEL
LIN {X 0,Y 143.785,Z 780.782,A -85,B 0,C 180,E1 -26055.006,E2 -26055.006} C_VEL
LIN {X 0,Y 145.682,Z 781.054,A -85,B 0,C 180,E1 -26055.67,E2 -26055.67} C_VEL
LIN {X 0,Y 145.12,Z 780.941,A -85,B 0,C 180,E1 -26056.403,E2 -26056.403} C_VEL
LIN {X 0,Y 138.725,Z 779.49,A -85,B 0,C 180,E1 -26058.807,E2 -26058.807} C_VEL
LIN {X 0,Y 133.943,Z 777.895,A -85,B 0,C 180,E1 -26060.976,E2 -26060.976} C_VEL
LIN {X 0,Y 127.496,Z 774.739,A -85,B 0,C 180,E1 -26064.634,E2 -26064.634} C_VEL
LIN {X 0,Y 122.05,Z 770.657,A -85,B 0,C 180,E1 -26068.785,E2 -26068.785} C_VEL
LIN {X 0,Y 117.673,Z 765.531,A -85,B 0,C 180,E1 -26073.627,E2 -26073.627} C_VEL
LIN {X 0,Y 114.457,Z 758.526,A -85,B 0,C 180,E1 -26079.452,E2 -26079.452} C_VEL
LIN {X 0,Y 113.078,Z 751.137,A -85,B 0,C 180,E1 -26084.684,E2 -26084.684} C_VEL
LIN {X 0,Y 112.925,Z 743.578,A -85,B 0,C 180,E1 -26089.239,E2 -26089.239} C_VEL
LIN {X 0,Y 113.164,Z 736.241,A -85,B 0,C 180,E1 -26092.865,E2 -26092.865} C_VEL
LIN {X 0,Y 113.266,Z 726.306,A -85,B 0,C 180,E1 -26096.443,E2 -26096.443} C_VEL
LIN {X 0,Y 113.131,Z 716.24,A -85,B 0,C 180,E1 -26099.11,E2 -26099.11} C_VEL
LIN {X 0,Y 112.994,Z 705.639,A -85,B 0,C 180,E1 -26101.345,E2 -26101.345} C_VEL
LIN {X 0,Y 112.536,Z 703.818,A -85,B 0,C 180,E1 -26102.195,E2 -26102.195} C_VEL
LIN {X 0,Y 112.236,Z 703.519,A -85,B 0,C 180,E1 -26102.92,E2 -26102.92} C_VEL
LIN {X 0,Y 112.218,Z 703.606,A -85,B 0,C 180,E1 -26103.591,E2 -26103.591} C_VEL
LIN {X 0,Y 112.883,Z 702.621,A -85,B 0,C 180,E1 -26104.999,E2 -26104.999} C_VEL
LIN {X 0,Y 114.509,Z 699.73,A -85,B 0,C 180,E1 -26106.519,E2 -26106.519} C_VEL
LIN {X 0,Y 115.266,Z 698.329,A -85,B 0,C 180,E1 -26107.005,E2 -26107.005} C_VEL
LIN {X 0,Y 116.114,Z 696.842,A -85,B 0,C 180,E1 -26107.827,E2 -26107.827} C_VEL
LIN {X 0,Y 117.746,Z 694.745,A -85,B 0,C 180,E1 -26110.315,E2 -26110.315} C_VEL
LIN {X 0,Y 119.557,Z 691.717,A -85,B 0,C 180,E1 -26111.84,E2 -26111.84} C_VEL
LIN {X 0,Y 122.151,Z 686.406,A -85,B 0,C 180,E1 -26113.306,E2 -26113.306} C_VEL
LIN {X 0,Y 122.975,Z 684.492,A -85,B 0,C 180,E1 -26113.69,E2 -26113.69} C_VEL
LIN {X 0,Y 125.88,Z 679.743,A -85,B 0,C 180,E1 -26116.314,E2 -26116.314} C_VEL
LIN {X 0,Y 128.335,Z 674.536,A -85,B 0,C 180,E1 -26117.941,E2 -26117.941} C_VEL
LIN {X 0,Y 131.048,Z 666.822,A -85,B 0,C 180,E1 -26119.38,E2 -26119.38} C_VEL
LIN {X 0,Y 132.649,Z 660.903,A -85,B 0,C 180,E1 -26120.245,E2 -26120.245} C_VEL
LIN {X 0,Y 135.032,Z 656.293,A -85,B 0,C 180,E1 -26122.226,E2 -26122.226} C_VEL
LIN {X 0,Y 137.588,Z 649.854,A -85,B 0,C 180,E1 -26123.919,E2 -26123.919} C_VEL
LIN {X 0,Y 141.04,Z 647.263,A -85,B 0,C 180,E1 -26126.646,E2 -26126.646} C_VEL
LIN {X 0,Y 145.208,Z 642.847,A -85,B 0,C 180,E1 -26129.348,E2 -26129.348} C_VEL
LIN {X 0,Y 148.244,Z 639.113,A -85,B 0,C 180,E1 -26131.046,E2 -26131.046} C_VEL
LIN {X 0,Y 152.963,Z 636.302,A -85,B 0,C 180,E1 -26133.657,E2 -26133.657} C_VEL
LIN {X 0,Y 155.372,Z 634.365,A -85,B 0,C 180,E1 -26134.825,E2 -26134.825} C_VEL
LIN {X 0,Y 155.882,Z 634.265,A -85,B 0,C 180,E1 -26135.089,E2 -26135.089} C_VEL
LIN {X 0,Y 157.035,Z 636.882,A -85,B 0,C 180,E1 -26135.89,E2 -26135.89} C_VEL
LIN {X 0,Y 154.493,Z 666.889,A -85,B 0,C 180,E1 -26137.032,E2 -26137.032} C_VEL
LIN {X 0,Y 152.388,Z 679.562,A -85,B 0,C 180,E1 -26137.825,E2 -26137.825} C_VEL
LIN {X 0,Y 149.401,Z 692.28,A -85,B 0,C 180,E1 -26139.085,E2 -26139.085} C_VEL
LIN {X 0,Y 145.812,Z 703.543,A -85,B 0,C 180,E1 -26140.609,E2 -26140.609} C_VEL
LIN {X 0,Y 141.101,Z 715.161,A -85,B 0,C 180,E1 -26142.717,E2 -26142.717} C_VEL
LIN {X 0,Y 136.046,Z 725.601,A -85,B 0,C 180,E1 -26145.26,E2 -26145.26} C_VEL
LIN {X 0,Y 131.34,Z 734.124,A -85,B 0,C 180,E1 -26148.017,E2 -26148.017} C_VEL
LIN {X 0,Y 126.815,Z 741.485,A -85,B 0,C 180,E1 -26151.089,E2 -26151.089} C_VEL
LIN {X 0,Y 122.076,Z 748.479,A -85,B 0,C 180,E1 -26154.847,E2 -26154.847} C_VEL
LIN {X 0,Y 117.256,Z 754.885,A -85,B 0,C 180,E1 -26159.368,E2 -26159.368} C_VEL
LIN {X 0,Y 113.191,Z 759.964,A -85,B 0,C 180,E1 -26164.235,E2 -26164.235} C_VEL
LIN {X 0,Y 109.93,Z 763.901,A -85,B 0,C 180,E1 -26169.41,E2 -26169.41} C_VEL
LIN {X 0,Y 107.564,Z 766.804,A -85,B 0,C 180,E1 -26174.846,E2 -26174.846} C_VEL
LIN {X 0,Y 105.746,Z 769.176,A -85,B 0,C 180,E1 -26182.358,E2 -26182.358} C_VEL
LIN {X 0,Y 105.344,Z 769.781,A -85,B 0,C 180,E1 -26186.171,E2 -26186.171} C_VEL
LIN {X 0,Y 105.238,Z 770.006,A -85,B 0,C 180,E1 -26189.997,E2 -26189.997} C_VEL
LIN {X 0,Y 105.343,Z 769.811,A -85,B 0,C 180,E1 -26193.822,E2 -26193.822} C_VEL
LIN {X 0,Y 105.744,Z 769.226,A -85,B 0,C 180,E1 -26197.635,E2 -26197.635} C_VEL
LIN {X 0,Y 107.559,Z 766.905,A -85,B 0,C 180,E1 -26205.147,E2 -26205.147} C_VEL
LIN {X 0,Y 109.9,Z 764.034,A -85,B 0,C 180,E1 -26210.589,E2 -26210.589} C_VEL
LIN {X 0,Y 113.115,Z 760.137,A -85,B 0,C 180,E1 -26215.776,E2 -26215.776} C_VEL
LIN {X 0,Y 117.176,Z 755.112,A -85,B 0,C 180,E1 -26220.648,E2 -26220.648} C_VEL
LIN {X 0,Y 122.005,Z 748.778,A -85,B 0,C 180,E1 -26225.169,E2 -26225.169} C_VEL
LIN {X 0,Y 127.55,Z 740.561,A -85,B 0,C 180,E1 -26229.52,E2 -26229.52} C_VEL
LIN {X 0,Y 133.313,Z 731,A -85,B 0,C 180,E1 -26233.258,E2 -26233.258} C_VEL
LIN {X 0,Y 138.753,Z 720.639,A -85,B 0,C 180,E1 -26236.197,E2 -26236.197} C_VEL
LIN {X 0,Y 143.321,Z 710.381,A -85,B 0,C 180,E1 -26238.397,E2 -26238.397} C_VEL
LIN {X 0,Y 147.485,Z 699.14,A -85,B 0,C 180,E1 -26240.206,E2 -26240.206} C_VEL
LIN {X 0,Y 150.823,Z 687.696,A -85,B 0,C 180,E1 -26241.571,E2 -26241.571} C_VEL
LIN {X 0,Y 153.552,Z 674.602,A -85,B 0,C 180,E1 -26242.668,E2 -26242.668} C_VEL
LIN {X 0,Y 155.307,Z 661.138,A -85,B 0,C 180,E1 -26243.367,E2 -26243.367} C_VEL
LIN {X 0,Y 157.229,Z 636.999,A -85,B 0,C 180,E1 -26244.256,E2 -26244.256} C_VEL
LIN {X 0,Y 152.633,Z 627.702,A -85,B 0,C 180,E1 -26247.54,E2 -26247.54} C_VEL
LIN {X 0,Y 148.455,Z 620.096,A -85,B 0,C 180,E1 -26250.928,E2 -26250.928} C_VEL
LIN {X 0,Y 144.251,Z 613.322,A -85,B 0,C 180,E1 -26254.888,E2 -26254.888} C_VEL
LIN {X 0,Y 141.907,Z 609.753,A -85,B 0,C 180,E1 -26257.469,E2 -26257.469} C_VEL
LIN {X 0,Y 138.919,Z 605.379,A -85,B 0,C 180,E1 -26261.376,E2 -26261.376} C_VEL
LIN {X 0,Y 136.56,Z 602.103,A -85,B 0,C 180,E1 -26265.279,E2 -26265.279} C_VEL
LIN {X 0,Y 135.963,Z 600.911,A -85,B 0,C 180,E1 -26266.549,E2 -26266.549} C_VEL
LIN {X 0,Y 133.461,Z 597.786,A -85,B 0,C 180,E1 -26273.765,E2 -26273.765} C_VEL
LIN {X 0,Y 133.027,Z 595.544,A -85,B 0,C 180,E1 -26278.486,E2 -26278.486} C_VEL
LIN {X 0,Y 133.042,Z 595.718,A -85,B 0,C 180,E1 -26281.703,E2 -26281.703} C_VEL
LIN {X 0,Y 135.419,Z 600.528,A -85,B 0,C 180,E1 -26291.981,E2 -26291.981} C_VEL
LIN {X 0,Y 136.215,Z 601.295,A -85,B 0,C 180,E1 -26293.615,E2 -26293.615} C_VEL
LIN {X 0,Y 138.3,Z 604.737,A -85,B 0,C 180,E1 -26297.37,E2 -26297.37} C_VEL
LIN {X 0,Y 139.516,Z 606.216,A -85,B 0,C 180,E1 -26299.113,E2 -26299.113} C_VEL
LIN {X 0,Y 142.719,Z 610.993,A -85,B 0,C 180,E1 -26303.105,E2 -26303.105} C_VEL
LIN {X 0,Y 145.536,Z 615.423,A -85,B 0,C 180,E1 -26306.049,E2 -26306.049} C_VEL
LIN {X 0,Y 147.66,Z 618.976,A -85,B 0,C 180,E1 -26308.035,E2 -26308.035} C_VEL
LIN {X 0,Y 151.362,Z 627.327,A -85,B 0,C 180,E1 -26311.296,E2 -26311.296} C_VEL
LIN {X 0,Y 155.127,Z 636.973,A -85,B 0,C 180,E1 -26314.28,E2 -26314.28} C_VEL
LIN {X 0,Y 156.885,Z 642.319,A -85,B 0,C 180,E1 -26315.617,E2 -26315.617} C_VEL
LIN {X 0,Y 154.258,Z 672.248,A -85,B 0,C 180,E1 -26316.712,E2 -26316.712} C_VEL
LIN {X 0,Y 151.925,Z 686.043,A -85,B 0,C 180,E1 -26317.595,E2 -26317.595} C_VEL
LIN {X 0,Y 148.725,Z 698.53,A -85,B 0,C 180,E1 -26318.771,E2 -26318.771} C_VEL
LIN {X 0,Y 144.942,Z 709.602,A -85,B 0,C 180,E1 -26320.214,E2 -26320.214} C_VEL
LIN {X 0,Y 140.106,Z 721.147,A -85,B 0,C 180,E1 -26322.282,E2 -26322.282} C_VEL
LIN {X 0,Y 134.984,Z 731.549,A -85,B 0,C 180,E1 -26324.819,E2 -26324.819} C_VEL
LIN {X 0,Y 130.09,Z 740.055,A -85,B 0,C 180,E1 -26327.527,E2 -26327.527} C_VEL
LIN {X 0,Y 124.188,Z 749.278,A -85,B 0,C 180,E1 -26331.504,E2 -26331.504} C_VEL
LIN {X 0,Y 118.65,Z 757.217,A -85,B 0,C 180,E1 -26336.23,E2 -26336.23} C_VEL
LIN {X 0,Y 114.507,Z 762.663,A -85,B 0,C 180,E1 -26340.597,E2 -26340.597} C_VEL
LIN {X 0,Y 110.829,Z 767.377,A -85,B 0,C 180,E1 -26345.662,E2 -26345.662} C_VEL
LIN {X 0,Y 107.989,Z 770.985,A -85,B 0,C 180,E1 -26351.014,E2 -26351.014} C_VEL
LIN {X 0,Y 106.704,Z 772.848,A -85,B 0,C 180,E1 -26354.728,E2 -26354.728} C_VEL
LIN {X 0,Y 105.796,Z 774.247,A -85,B 0,C 180,E1 -26358.508,E2 -26358.508} C_VEL
LIN {X 0,Y 105.035,Z 775.857,A -85,B 0,C 180,E1 -26366.167,E2 -26366.167} C_VEL
LIN {X 0,Y 105.168,Z 776.073,A -85,B 0,C 180,E1 -26370.003,E2 -26370.003} C_VEL
LIN {X 0,Y 105.343,Z 775.848,A -85,B 0,C 180,E1 -26373.829,E2 -26373.829} C_VEL
LIN {X 0,Y 106.766,Z 774.23,A -85,B 0,C 180,E1 -26381.393,E2 -26381.393} C_VEL
LIN {X 0,Y 108.061,Z 772.826,A -85,B 0,C 180,E1 -26385.082,E2 -26385.082} C_VEL
LIN {X 0,Y 111.135,Z 769.898,A -85,B 0,C 180,E1 -26390.357,E2 -26390.357} C_VEL
LIN {X 0,Y 116.209,Z 765.408,A -85,B 0,C 180,E1 -26396.009,E2 -26396.009} C_VEL
LIN {X 0,Y 116.841,Z 765.957,A -85,B 0,C 180,E1 -26396.819,E2 -26396.819} C_VEL
LIN {X 0,Y 120.676,Z 770.579,A -85,B 0,C 180,E1 -26401.614,E2 -26401.614} C_VEL
LIN {X 0,Y 124.14,Z 773.441,A -85,B 0,C 180,E1 -26404.742,E2 -26404.742} C_VEL
LIN {X 0,Y 125.634,Z 774.501,A -85,B 0,C 180,E1 -26406.369,E2 -26406.369} C_VEL
LIN {X 0,Y 128.589,Z 776.463,A -85,B 0,C 180,E1 -26412.246,E2 -26412.246} C_VEL
LIN {X 0,Y 130.662,Z 777.222,A -85,B 0,C 180,E1 -26413.7,E2 -26413.7} C_VEL
LIN {X 0,Y 133.513,Z 778.252,A -85,B 0,C 180,E1 -26414.983,E2 -26414.983} C_VEL
LIN {X 0,Y 134.666,Z 778.572,A -85,B 0,C 180,E1 -26416.381,E2 -26416.381} C_VEL
LIN {X 0,Y 126.361,Z 775.118,A -85,B 0,C 180,E1 -26420.237,E2 -26420.237} C_VEL
LIN {X 0,Y 120.038,Z 771.154,A -85,B 0,C 180,E1 -26424.163,E2 -26424.163} C_VEL
LIN {X 0,Y 114.701,Z 766.163,A -85,B 0,C 180,E1 -26428.819,E2 -26428.819} C_VEL
LIN {X 0,Y 109.927,Z 758.544,A -85,B 0,C 180,E1 -26435.445,E2 -26435.445} C_VEL
LIN {X 0,Y 107.891,Z 751.137,A -85,B 0,C 180,E1 -26440.992,E2 -26440.992} C_VEL
LIN {X 0,Y 107.212,Z 743.892,A -85,B 0,C 180,E1 -26445.77,E2 -26445.77} C_VEL
LIN {X 0,Y 107.323,Z 736.878,A -85,B 0,C 180,E1 -26449.624,E2 -26449.624} C_VEL
LIN {X 0,Y 107.409,Z 730.389,A -85,B 0,C 180,E1 -26452.481,E2 -26452.481} C_VEL
LIN {X 0,Y 107.322,Z 722.508,A -85,B 0,C 180,E1 -26455.211,E2 -26455.211} C_VEL
LIN {X 0,Y 107,Z 715.862,A -85,B 0,C 180,E1 -26457.177,E2 -26457.177} C_VEL
LIN {X 0,Y 106.403,Z 714.416,A -85,B 0,C 180,E1 -26458.226,E2 -26458.226} C_VEL
LIN {X 0,Y 106.077,Z 714.324,A -85,B 0,C 180,E1 -26460,E2 -26460} C_VEL
LIN {X 0,Y 106.523,Z 713.546,A -85,B 0,C 180,E1 -26461.182,E2 -26461.182} C_VEL
LIN {X 0,Y 108.109,Z 711.073,A -85,B 0,C 180,E1 -26463.006,E2 -26463.006} C_VEL
LIN {X 0,Y 108.871,Z 709.861,A -85,B 0,C 180,E1 -26463.701,E2 -26463.701} C_VEL
LIN {X 0,Y 109.334,Z 709.346,A -85,B 0,C 180,E1 -26465.161,E2 -26465.161} C_VEL
LIN {X 0,Y 110.648,Z 707.649,A -85,B 0,C 180,E1 -26467.298,E2 -26467.298} C_VEL
LIN {X 0,Y 113.458,Z 703.448,A -85,B 0,C 180,E1 -26469.499,E2 -26469.499} C_VEL
LIN {X 0,Y 114.196,Z 702.313,A -85,B 0,C 180,E1 -26470.023,E2 -26470.023} C_VEL
LIN {X 0,Y 115.956,Z 700.368,A -85,B 0,C 180,E1 -26472.248,E2 -26472.248} C_VEL
LIN {X 0,Y 118.497,Z 696.823,A -85,B 0,C 180,E1 -26474.218,E2 -26474.218} C_VEL
LIN {X 0,Y 121.046,Z 692.541,A -85,B 0,C 180,E1 -26475.583,E2 -26475.583} C_VEL
LIN {X 0,Y 123.198,Z 688.522,A -85,B 0,C 180,E1 -26476.573,E2 -26476.573} C_VEL
LIN {X 0,Y 126.249,Z 684.156,A -85,B 0,C 180,E1 -26478.845,E2 -26478.845} C_VEL
LIN {X 0,Y 129.223,Z 678.658,A -85,B 0,C 180,E1 -26480.495,E2 -26480.495} C_VEL
LIN {X 0,Y 132.388,Z 670.891,A -85,B 0,C 180,E1 -26481.917,E2 -26481.917} C_VEL
LIN {X 0,Y 134.331,Z 665.08,A -85,B 0,C 180,E1 -26482.798,E2 -26482.798} C_VEL
LIN {X 0,Y 136.971,Z 660.168,A -85,B 0,C 180,E1 -26484.639,E2 -26484.639} C_VEL
LIN {X 0,Y 138.734,Z 655.973,A -85,B 0,C 180,E1 -26485.707,E2 -26485.707} C_VEL
LIN {X 0,Y 143.008,Z 652.452,A -85,B 0,C 180,E1 -26488.731,E2 -26488.731} C_VEL
LIN {X 0,Y 148.358,Z 646.602,A -85,B 0,C 180,E1 -26491.804,E2 -26491.804} C_VEL
LIN {X 0,Y 149.4,Z 645.495,A -85,B 0,C 180,E1 -26492.351,E2 -26492.351} C_VEL
LIN {X 0,Y 152.45,Z 643.717,A -85,B 0,C 180,E1 -26493.985,E2 -26493.985} C_VEL
LIN {X 0,Y 150.221,Z 667.911,A -85,B 0,C 180,E1 -26494.918,E2 -26494.918} C_VEL
LIN {X 0,Y 147.988,Z 680.556,A -85,B 0,C 180,E1 -26495.723,E2 -26495.723} C_VEL
LIN {X 0,Y 144.715,Z 693.565,A -85,B 0,C 180,E1 -26497.031,E2 -26497.031} C_VEL
LIN {X 0,Y 141.299,Z 703.752,A -85,B 0,C 180,E1 -26498.425,E2 -26498.425} C_VEL
LIN {X 0,Y 136.397,Z 715.37,A -85,B 0,C 180,E1 -26500.532,E2 -26500.532} C_VEL
LIN {X 0,Y 131.114,Z 725.808,A -85,B 0,C 180,E1 -26503.082,E2 -26503.082} C_VEL
LIN {X 0,Y 126.147,Z 734.331,A -85,B 0,C 180,E1 -26505.857,E2 -26505.857} C_VEL
LIN {X 0,Y 121.038,Z 742.192,A -85,B 0,C 180,E1 -26509.218,E2 -26509.218} C_VEL
LIN {X 0,Y 115.458,Z 749.849,A -85,B 0,C 180,E1 -26513.591,E2 -26513.591} C_VEL
LIN {X 0,Y 109.61,Z 756.899,A -85,B 0,C 180,E1 -26519.136,E2 -26519.136} C_VEL
LIN {X 0,Y 105.591,Z 761.584,A -85,B 0,C 180,E1 -26524.362,E2 -26524.362} C_VEL
LIN {X 0,Y 102.341,Z 765.164,A -85,B 0,C 180,E1 -26529.915,E2 -26529.915} C_VEL
LIN {X 0,Y 100.717,Z 767.01,A -85,B 0,C 180,E1 -26533.789,E2 -26533.789} C_VEL
LIN {X 0,Y 99.514,Z 768.396,A -85,B 0,C 180,E1 -26537.764,E2 -26537.764} C_VEL
LIN {X 0,Y 98.704,Z 769.381,A -85,B 0,C 180,E1 -26541.809,E2 -26541.809} C_VEL
LIN {X 0,Y 98.26,Z 769.986,A -85,B 0,C 180,E1 -26545.895,E2 -26545.895} C_VEL
LIN {X 0,Y 98.152,Z 770.21,A -85,B 0,C 180,E1 -26549.996,E2 -26549.996} C_VEL
LIN {X 0,Y 98.259,Z 770.015,A -85,B 0,C 180,E1 -26554.098,E2 -26554.098} C_VEL
LIN {X 0,Y 98.702,Z 769.431,A -85,B 0,C 180,E1 -26558.183,E2 -26558.183} C_VEL
LIN {X 0,Y 100.709,Z 767.109,A -85,B 0,C 180,E1 -26566.205,E2 -26566.205} C_VEL
LIN {X 0,Y 103.287,Z 764.238,A -85,B 0,C 180,E1 -26571.973,E2 -26571.973} C_VEL
LIN {X 0,Y 106.748,Z 760.341,A -85,B 0,C 180,E1 -26577.439,E2 -26577.439} C_VEL
LIN {X 0,Y 111.134,Z 755.315,A -85,B 0,C 180,E1 -26582.512,E2 -26582.512} C_VEL
LIN {X 0,Y 116.267,Z 748.981,A -85,B 0,C 180,E1 -26587.187,E2 -26587.187} C_VEL
LIN {X 0,Y 121.832,Z 741.243,A -85,B 0,C 180,E1 -26591.416,E2 -26591.416} C_VEL
LIN {X 0,Y 127.151,Z 732.98,A -85,B 0,C 180,E1 -26594.803,E2 -26594.803} C_VEL
LIN {X 0,Y 132.751,Z 723.116,A -85,B 0,C 180,E1 -26597.827,E2 -26597.827} C_VEL
LIN {X 0,Y 138.122,Z 712.002,A -85,B 0,C 180,E1 -26600.313,E2 -26600.313} C_VEL
LIN {X 0,Y 142.439,Z 701.101,A -85,B 0,C 180,E1 -26602.129,E2 -26602.129} C_VEL
LIN {X 0,Y 146.2,Z 689.038,A -85,B 0,C 180,E1 -26603.624,E2 -26603.624} C_VEL
LIN {X 0,Y 149.032,Z 676.699,A -85,B 0,C 180,E1 -26604.705,E2 -26604.705} C_VEL
LIN {X 0,Y 150.992,Z 663.181,A -85,B 0,C 180,E1 -26605.448,E2 -26605.448} C_VEL
LIN {X 0,Y 152.946,Z 639.957,A -85,B 0,C 180,E1 -26606.319,E2 -26606.319} C_VEL
LIN {X 0,Y 148.554,Z 630.882,A -85,B 0,C 180,E1 -26609.82,E2 -26609.82} C_VEL
LIN {X 0,Y 144.82,Z 623.955,A -85,B 0,C 180,E1 -26613.23,E2 -26613.23} C_VEL
LIN {X 0,Y 141.381,Z 618.336,A -85,B 0,C 180,E1 -26616.873,E2 -26616.873} C_VEL
LIN {X 0,Y 139.898,Z 615.962,A -85,B 0,C 180,E1 -26618.681,E2 -26618.681} C_VEL
LIN {X 0,Y 137.336,Z 611.978,A -85,B 0,C 180,E1 -26622.311,E2 -26622.311} C_VEL
LIN {X 0,Y 135.062,Z 608.459,A -85,B 0,C 180,E1 -26626.458,E2 -26626.458} C_VEL
LIN {X 0,Y 134.572,Z 607.671,A -85,B 0,C 180,E1 -26627.559,E2 -26627.559} C_VEL
LIN {X 0,Y 132.147,Z 602.803,A -85,B 0,C 180,E1 -26638.288,E2 -26638.288} C_VEL
LIN {X 0,Y 132.143,Z 602.56,A -85,B 0,C 180,E1 -26640.627,E2 -26640.627} C_VEL
LIN {X 0,Y 134.958,Z 608.176,A -85,B 0,C 180,E1 -26652.93,E2 -26652.93} C_VEL
LIN {X 0,Y 137.071,Z 611.683,A -85,B 0,C 180,E1 -26656.922,E2 -26656.922} C_VEL
LIN {X 0,Y 138.126,Z 613.256,A -85,B 0,C 180,E1 -26658.542,E2 -26658.542} C_VEL
LIN {X 0,Y 140.947,Z 617.596,A -85,B 0,C 180,E1 -26662.25,E2 -26662.25} C_VEL
LIN {X 0,Y 143.625,Z 622.013,A -85,B 0,C 180,E1 -26665.22,E2 -26665.22} C_VEL
LIN {X 0,Y 145.427,Z 625.413,A -85,B 0,C 180,E1 -26667.038,E2 -26667.038} C_VEL
LIN {X 0,Y 149.135,Z 634.454,A -85,B 0,C 180,E1 -26670.535,E2 -26670.535} C_VEL
LIN {X 0,Y 152.195,Z 643.232,A -85,B 0,C 180,E1 -26673.167,E2 -26673.167} C_VEL
LIN {X 0,Y 152.634,Z 644.725,A -85,B 0,C 180,E1 -26673.541,E2 -26673.541} C_VEL
LIN {X 0,Y 150.052,Z 672.544,A -85,B 0,C 180,E1 -26674.564,E2 -26674.564} C_VEL
LIN {X 0,Y 147.608,Z 686.276,A -85,B 0,C 180,E1 -26675.444,E2 -26675.444} C_VEL
LIN {X 0,Y 144.388,Z 698.332,A -85,B 0,C 180,E1 -26676.575,E2 -26676.575} C_VEL
LIN {X 0,Y 140.468,Z 709.403,A -85,B 0,C 180,E1 -26678.004,E2 -26678.004} C_VEL
LIN {X 0,Y 135.431,Z 720.946,A -85,B 0,C 180,E1 -26680.059,E2 -26680.059} C_VEL
LIN {X 0,Y 130.067,Z 731.347,A -85,B 0,C 180,E1 -26682.595,E2 -26682.595} C_VEL
LIN {X 0,Y 124.937,Z 739.853,A -85,B 0,C 180,E1 -26685.324,E2 -26685.324} C_VEL
LIN {X 0,Y 119.678,Z 747.702,A -85,B 0,C 180,E1 -26688.655,E2 -26688.655} C_VEL
LIN {X 0,Y 114.162,Z 755.261,A -85,B 0,C 180,E1 -26693.004,E2 -26693.004} C_VEL
LIN {X 0,Y 109.968,Z 760.641,A -85,B 0,C 180,E1 -26697.1,E2 -26697.1} C_VEL
LIN {X 0,Y 105.622,Z 765.738,A -85,B 0,C 180,E1 -26702.244,E2 -26702.244} C_VEL
LIN {X 0,Y 102.184,Z 769.704,A -85,B 0,C 180,E1 -26707.777,E2 -26707.777} C_VEL
LIN {X 0,Y 99.829,Z 772.643,A -85,B 0,C 180,E1 -26713.648,E2 -26713.648} C_VEL
LIN {X 0,Y 98.811,Z 774.041,A -85,B 0,C 180,E1 -26717.684,E2 -26717.684} C_VEL
LIN {X 0,Y 98.185,Z 775.041,A -85,B 0,C 180,E1 -26721.773,E2 -26721.773} C_VEL
LIN {X 0,Y 97.941,Z 775.652,A -85,B 0,C 180,E1 -26725.889,E2 -26725.889} C_VEL
LIN {X 0,Y 98.074,Z 775.869,A -85,B 0,C 180,E1 -26730.004,E2 -26730.004} C_VEL
LIN {X 0,Y 98.261,Z 775.643,A -85,B 0,C 180,E1 -26734.105,E2 -26734.105} C_VEL
LIN {X 0,Y 99.818,Z 774.025,A -85,B 0,C 180,E1 -26742.198,E2 -26742.198} C_VEL
LIN {X 0,Y 101.245,Z 772.621,A -85,B 0,C 180,E1 -26746.124,E2 -26746.124} C_VEL
LIN {X 0,Y 104.514,Z 769.693,A -85,B 0,C 180,E1 -26751.71,E2 -26751.71} C_VEL
LIN {X 0,Y 108.986,Z 765.717,A -85,B 0,C 180,E1 -26756.837,E2 -26756.837} C_VEL
LIN {X 0,Y 111.514,Z 763.803,A -85,B 0,C 180,E1 -26758.983,E2 -26758.983} C_VEL
LIN {X 0,Y 112.405,Z 764.551,A -85,B 0,C 180,E1 -26760.016,E2 -26760.016} C_VEL
LIN {X 0,Y 118.49,Z 770.767,A -85,B 0,C 180,E1 -26766.383,E2 -26766.383} C_VEL
LIN {X 0,Y 126.694,Z 775.666,A -85,B 0,C 180,E1 -26771.737,E2 -26771.737} C_VEL
LIN {X 0,Y 130.662,Z 777.222,A -85,B 0,C 180,E1 -26773.7,E2 -26773.7} C_VEL
LIN {X 0,Y 131.09,Z 777.4,A -85,B 0,C 180,E1 -26774.29,E2 -26774.29} C_VEL
LIN {X 0,Y 130.336,Z 777.14,A -85,B 0,C 180,E1 -26775.369,E2 -26775.369} C_VEL
LIN {X 0,Y 128.042,Z 776.224,A -85,B 0,C 180,E1 -26776.603,E2 -26776.603} C_VEL
LIN {X 0,Y 119.281,Z 771.756,A -85,B 0,C 180,E1 -26779.495,E2 -26779.495} C_VEL
LIN {X 0,Y 117.113,Z 770.287,A -85,B 0,C 180,E1 -26780.606,E2 -26780.606} C_VEL
LIN {X 0,Y 110.635,Z 764.676,A -85,B 0,C 180,E1 -26785.676,E2 -26785.676} C_VEL
LIN {X 0,Y 105.441,Z 756.996,A -85,B 0,C 180,E1 -26792.188,E2 -26792.188} C_VEL
LIN {X 0,Y 102.863,Z 749.659,A -85,B 0,C 180,E1 -26797.927,E2 -26797.927} C_VEL
LIN {X 0,Y 101.757,Z 739.689,A -85,B 0,C 180,E1 -26804.611,E2 -26804.611} C_VEL
LIN {X 0,Y 101.771,Z 733.484,A -85,B 0,C 180,E1 -26808.044,E2 -26808.044} C_VEL
LIN {X 0,Y 101.78,Z 727.868,A -85,B 0,C 180,E1 -26810.56,E2 -26810.56} C_VEL
LIN {X 0,Y 101.627,Z 725.187,A -85,B 0,C 180,E1 -26811.674,E2 -26811.674} C_VEL
LIN {X 0,Y 100.951,Z 723.687,A -85,B 0,C 180,E1 -26812.923,E2 -26812.923} C_VEL
LIN {X 0,Y 100.331,Z 723.57,A -85,B 0,C 180,E1 -26814.428,E2 -26814.428} C_VEL
LIN {X 0,Y 100.381,Z 723.125,A -85,B 0,C 180,E1 -26815.985,E2 -26815.985} C_VEL
LIN {X 0,Y 101.402,Z 721.404,A -85,B 0,C 180,E1 -26818.014,E2 -26818.014} C_VEL
LIN {X 0,Y 102.132,Z 720.235,A -85,B 0,C 180,E1 -26820,E2 -26820} C_VEL
LIN {X 0,Y 102.632,Z 719.486,A -85,B 0,C 180,E1 -26821.962,E2 -26821.962} C_VEL
LIN {X 0,Y 103.81,Z 717.913,A -85,B 0,C 180,E1 -26823.882,E2 -26823.882} C_VEL
LIN {X 0,Y 105.805,Z 715.324,A -85,B 0,C 180,E1 -26825.91,E2 -26825.91} C_VEL
LIN {X 0,Y 108.029,Z 712.946,A -85,B 0,C 180,E1 -26829.36,E2 -26829.36} C_VEL
LIN {X 0,Y 110.857,Z 709.456,A -85,B 0,C 180,E1 -26831.532,E2 -26831.532} C_VEL
LIN {X 0,Y 112.491,Z 707.296,A -85,B 0,C 180,E1 -26832.631,E2 -26832.631} C_VEL
LIN {X 0,Y 114.038,Z 705.841,A -85,B 0,C 180,E1 -26834.272,E2 -26834.272} C_VEL
LIN {X 0,Y 117.355,Z 701.893,A -85,B 0,C 180,E1 -26836.617,E2 -26836.617} C_VEL
LIN {X 0,Y 120.69,Z 697.1,A -85,B 0,C 180,E1 -26838.24,E2 -26838.24} C_VEL
LIN {X 0,Y 123.281,Z 692.937,A -85,B 0,C 180,E1 -26839.316,E2 -26839.316} C_VEL
LIN {X 0,Y 126.346,Z 688.987,A -85,B 0,C 180,E1 -26841.196,E2 -26841.196} C_VEL
LIN {X 0,Y 130.235,Z 682.671,A -85,B 0,C 180,E1 -26843.042,E2 -26843.042} C_VEL
LIN {X 0,Y 134.014,Z 674.542,A -85,B 0,C 180,E1 -26844.465,E2 -26844.465} C_VEL
LIN {X 0,Y 136.052,Z 669.286,A -85,B 0,C 180,E1 -26845.225,E2 -26845.225} C_VEL
LIN {X 0,Y 139.04,Z 664.081,A -85,B 0,C 180,E1 -26846.958,E2 -26846.958} C_VEL
LIN {X 0,Y 140.243,Z 661.735,A -85,B 0,C 180,E1 -26847.616,E2 -26847.616} C_VEL
LIN {X 0,Y 144.803,Z 657.868,A -85,B 0,C 180,E1 -26850.538,E2 -26850.538} C_VEL
LIN {X 0,Y 147.621,Z 654.956,A -85,B 0,C 180,E1 -26852.098,E2 -26852.098} C_VEL
LIN {X 0,Y 145.917,Z 670.611,A -85,B 0,C 180,E1 -26852.767,E2 -26852.767} C_VEL
LIN {X 0,Y 143.445,Z 683.014,A -85,B 0,C 180,E1 -26853.598,E2 -26853.598} C_VEL
LIN {X 0,Y 140.222,Z 694.769,A -85,B 0,C 180,E1 -26854.839,E2 -26854.839} C_VEL
LIN {X 0,Y 135.758,Z 707.118,A -85,B 0,C 180,E1 -26856.635,E2 -26856.635} C_VEL
LIN {X 0,Y 130.659,Z 718.142,A -85,B 0,C 180,E1 -26858.741,E2 -26858.741} C_VEL
LIN {X 0,Y 125.76,Z 727.071,A -85,B 0,C 180,E1 -26861.02,E2 -26861.02} C_VEL
LIN {X 0,Y 120.031,Z 736.224,A -85,B 0,C 180,E1 -26864.168,E2 -26864.168} C_VEL
LIN {X 0,Y 113.695,Z 745.119,A -85,B 0,C 180,E1 -26868.352,E2 -26868.352} C_VEL
LIN {X 0,Y 107.958,Z 752.276,A -85,B 0,C 180,E1 -26872.971,E2 -26872.971} C_VEL
LIN {X 0,Y 103.589,Z 757.105,A -85,B 0,C 180,E1 -26877.124,E2 -26877.124} C_VEL
LIN {X 0,Y 99.24,Z 761.79,A -85,B 0,C 180,E1 -26882.588,E2 -26882.588} C_VEL
LIN {X 0,Y 95.702,Z 765.369,A -85,B 0,C 180,E1 -26888.454,E2 -26888.454} C_VEL
LIN {X 0,Y 93.918,Z 767.215,A -85,B 0,C 180,E1 -26892.579,E2 -26892.579} C_VEL
LIN {X 0,Y 92.582,Z 768.601,A -85,B 0,C 180,E1 -26896.832,E2 -26896.832} C_VEL
LIN {X 0,Y 91.694,Z 769.586,A -85,B 0,C 180,E1 -26901.178,E2 -26901.178} C_VEL
LIN {X 0,Y 91.205,Z 770.19,A -85,B 0,C 180,E1 -26905.577,E2 -26905.577} C_VEL
LIN {X 0,Y 91.058,Z 770.415,A -85,B 0,C 180,E1 -26909.996,E2 -26909.996} C_VEL
LIN {X 0,Y 91.185,Z 770.219,A -85,B 0,C 180,E1 -26914.416,E2 -26914.416} C_VEL
LIN {X 0,Y 91.692,Z 769.635,A -85,B 0,C 180,E1 -26918.814,E2 -26918.814} C_VEL
LIN {X 0,Y 93.91,Z 767.313,A -85,B 0,C 180,E1 -26927.414,E2 -26927.414} C_VEL
LIN {X 0,Y 96.749,Z 764.441,A -85,B 0,C 180,E1 -26933.544,E2 -26933.544} C_VEL
LIN {X 0,Y 100.484,Z 760.545,A -85,B 0,C 180,E1 -26939.309,E2 -26939.309} C_VEL
LIN {X 0,Y 105.224,Z 755.518,A -85,B 0,C 180,E1 -26944.587,E2 -26944.587} C_VEL
LIN {X 0,Y 110.686,Z 749.184,A -85,B 0,C 180,E1 -26949.412,E2 -26949.412} C_VEL
LIN {X 0,Y 116.892,Z 741.013,A -85,B 0,C 180,E1 -26953.938,E2 -26953.938} C_VEL
LIN {X 0,Y 123.362,Z 731.404,A -85,B 0,C 180,E1 -26957.779,E2 -26957.779} C_VEL
LIN {X 0,Y 128.73,Z 722.211,A -85,B 0,C 180,E1 -26960.453,E2 -26960.453} C_VEL
LIN {X 0,Y 134.337,Z 710.78,A -85,B 0,C 180,E1 -26962.917,E2 -26962.917} C_VEL
LIN {X 0,Y 138.849,Z 699.536,A -85,B 0,C 180,E1 -26964.7,E2 -26964.7} C_VEL
LIN {X 0,Y 142.438,Z 688.09,A -85,B 0,C 180,E1 -26966.047,E2 -26966.047} C_VEL
LIN {X 0,Y 145.465,Z 674.663,A -85,B 0,C 180,E1 -26967.127,E2 -26967.127} C_VEL
LIN {X 0,Y 147.339,Z 661.132,A -85,B 0,C 180,E1 -26967.806,E2 -26967.806} C_VEL
LIN {X 0,Y 148.903,Z 643.106,A -85,B 0,C 180,E1 -26968.46,E2 -26968.46} C_VEL
LIN {X 0,Y 144.877,Z 634.473,A -85,B 0,C 180,E1 -26972.068,E2 -26972.068} C_VEL
LIN {X 0,Y 141.488,Z 628.159,A -85,B 0,C 180,E1 -26975.553,E2 -26975.553} C_VEL
LIN {X 0,Y 138.244,Z 622.542,A -85,B 0,C 180,E1 -26979.542,E2 -26979.542} C_VEL
LIN {X 0,Y 135.791,Z 618.572,A -85,B 0,C 180,E1 -26983.268,E2 -26983.268} C_VEL
LIN {X 0,Y 133.428,Z 614.54,A -85,B 0,C 180,E1 -26988.126,E2 -26988.126} C_VEL
LIN {X 0,Y 131.274,Z 609.576,A -85,B 0,C 180,E1 -26999.282,E2 -26999.282} C_VEL
LIN {X 0,Y 131.261,Z 609.972,A -85,B 0,C 180,E1 -27001.262,E2 -27001.262} C_VEL
LIN {X 0,Y 133.684,Z 614.972,A -85,B 0,C 180,E1 -27012.139,E2 -27012.139} C_VEL
LIN {X 0,Y 136.464,Z 619.654,A -85,B 0,C 180,E1 -27017.482,E2 -27017.482} C_VEL
LIN {X 0,Y 139.005,Z 623.865,A -85,B 0,C 180,E1 -27021.115,E2 -27021.115} C_VEL
LIN {X 0,Y 142.181,Z 629.349,A -85,B 0,C 180,E1 -27024.838,E2 -27024.838} C_VEL
LIN {X 0,Y 145.19,Z 636.976,A -85,B 0,C 180,E1 -27028.063,E2 -27028.063} C_VEL
LIN {X 0,Y 148.176,Z 645.682,A -85,B 0,C 180,E1 -27030.952,E2 -27030.952} C_VEL
LIN {X 0,Y 148.597,Z 647.115,A -85,B 0,C 180,E1 -27031.349,E2 -27031.349} C_VEL
LIN {X 0,Y 146.16,Z 672.218,A -85,B 0,C 180,E1 -27032.263,E2 -27032.263} C_VEL
LIN {X 0,Y 143.665,Z 685.774,A -85,B 0,C 180,E1 -27033.106,E2 -27033.106} C_VEL
LIN {X 0,Y 140.271,Z 698.134,A -85,B 0,C 180,E1 -27034.244,E2 -27034.244} C_VEL
LIN {X 0,Y 136.208,Z 709.203,A -85,B 0,C 180,E1 -27035.649,E2 -27035.649} C_VEL
LIN {X 0,Y 130.978,Z 720.746,A -85,B 0,C 180,E1 -27037.684,E2 -27037.684} C_VEL
LIN {X 0,Y 125.354,Z 731.145,A -85,B 0,C 180,E1 -27040.197,E2 -27040.197} C_VEL
LIN {X 0,Y 119.991,Z 739.651,A -85,B 0,C 180,E1 -27042.939,E2 -27042.939} C_VEL
LIN {X 0,Y 113.377,Z 748.872,A -85,B 0,C 180,E1 -27047.015,E2 -27047.015} C_VEL
LIN {X 0,Y 107.175,Z 756.692,A -85,B 0,C 180,E1 -27051.896,E2 -27051.896} C_VEL
LIN {X 0,Y 102.358,Z 762.256,A -85,B 0,C 180,E1 -27056.686,E2 -27056.686} C_VEL
LIN {X 0,Y 98.005,Z 766.968,A -85,B 0,C 180,E1 -27062.222,E2 -27062.222} C_VEL
LIN {X 0,Y 94.595,Z 770.575,A -85,B 0,C 180,E1 -27068.198,E2 -27068.198} C_VEL
LIN {X 0,Y 93.003,Z 772.438,A -85,B 0,C 180,E1 -27072.41,E2 -27072.41} C_VEL
LIN {X 0,Y 91.861,Z 773.836,A -85,B 0,C 180,E1 -27076.735,E2 -27076.735} C_VEL
LIN {X 0,Y 90.871,Z 775.448,A -85,B 0,C 180,E1 -27085.568,E2 -27085.568} C_VEL
LIN {X 0,Y 90.972,Z 775.664,A -85,B 0,C 180,E1 -27090.004,E2 -27090.004} C_VEL
LIN {X 0,Y 91.209,Z 775.439,A -85,B 0,C 180,E1 -27094.423,E2 -27094.423} C_VEL
LIN {X 0,Y 92.909,Z 773.82,A -85,B 0,C 180,E1 -27103.12,E2 -27103.12} C_VEL
LIN {X 0,Y 94.453,Z 772.416,A -85,B 0,C 180,E1 -27107.319,E2 -27107.319} C_VEL
LIN {X 0,Y 97.969,Z 769.488,A -85,B 0,C 180,E1 -27113.242,E2 -27113.242} C_VEL
LIN {X 0,Y 102.711,Z 765.521,A -85,B 0,C 180,E1 -27118.622,E2 -27118.622} C_VEL
LIN {X 0,Y 107.205,Z 762.07,A -85,B 0,C 180,E1 -27122.188,E2 -27122.188} C_VEL
LIN {X 0,Y 108.049,Z 762.579,A -85,B 0,C 180,E1 -27123.011,E2 -27123.011} C_VEL
LIN {X 0,Y 113.308,Z 767.938,A -85,B 0,C 180,E1 -27128.339,E2 -27128.339} C_VEL
LIN {X 0,Y 121.764,Z 773.403,A -85,B 0,C 180,E1 -27133.842,E2 -27133.842} C_VEL
LIN {X 0,Y 123.789,Z 774.35,A -85,B 0,C 180,E1 -27134.873,E2 -27134.873} C_VEL
LIN {X 0,Y 124.768,Z 774.754,A -85,B 0,C 180,E1 -27136.407,E2 -27136.407} C_VEL
LIN {X 0,Y 117.113,Z 770.287,A -85,B 0,C 180,E1 -27140.606,E2 -27140.606} C_VEL
LIN {X 0,Y 113.589,Z 767.675,A -85,B 0,C 180,E1 -27142.562,E2 -27142.562} C_VEL
LIN {X 0,Y 107.392,Z 762.22,A -85,B 0,C 180,E1 -27145.429,E2 -27145.429} C_VEL
LIN {X 0,Y 102.036,Z 756.193,A -85,B 0,C 180,E1 -27148.576,E2 -27148.576} C_VEL
LIN {X 0,Y 99.95,Z 752.614,A -85,B 0,C 180,E1 -27150.961,E2 -27150.961} C_VEL
LIN {X 0,Y 97.278,Z 743.703,A -85,B 0,C 180,E1 -27157.71,E2 -27157.71} C_VEL
LIN {X 0,Y 96.281,Z 734.309,A -85,B 0,C 180,E1 -27164.028,E2 -27164.028} C_VEL
LIN {X 0,Y 95.596,Z 732.918,A -85,B 0,C 180,E1 -27165.585,E2 -27165.585} C_VEL
LIN {X 0,Y 94.876,Z 732.749,A -85,B 0,C 180,E1 -27167.16,E2 -27167.16} C_VEL
LIN {X 0,Y 94.754,Z 732.056,A -85,B 0,C 180,E1 -27169.154,E2 -27169.154} C_VEL
LIN {X 0,Y 95.364,Z 730.545,A -85,B 0,C 180,E1 -27171.524,E2 -27171.524} C_VEL
LIN {X 0,Y 96.329,Z 727.928,A -85,B 0,C 180,E1 -27177.91,E2 -27177.91} C_VEL
LIN {X 0,Y 97.504,Z 726.316,A -85,B 0,C 180,E1 -27180,E2 -27180} C_VEL
LIN {X 0,Y 99.112,Z 724.419,A -85,B 0,C 180,E1 -27184.066,E2 -27184.066} C_VEL
LIN {X 0,Y 101.419,Z 721.85,A -85,B 0,C 180,E1 -27186.974,E2 -27186.974} C_VEL
LIN {X 0,Y 102.427,Z 720.745,A -85,B 0,C 180,E1 -27187.888,E2 -27187.888} C_VEL
LIN {X 0,Y 105.323,Z 718.059,A -85,B 0,C 180,E1 -27191.548,E2 -27191.548} C_VEL
LIN {X 0,Y 108.984,Z 714.153,A -85,B 0,C 180,E1 -27194.14,E2 -27194.14} C_VEL
LIN {X 0,Y 110.12,Z 712.83,A -85,B 0,C 180,E1 -27194.791,E2 -27194.791} C_VEL
LIN {X 0,Y 113.194,Z 710.008,A -85,B 0,C 180,E1 -27197.247,E2 -27197.247} C_VEL
LIN {X 0,Y 116.717,Z 706.228,A -85,B 0,C 180,E1 -27199.341,E2 -27199.341} C_VEL
LIN {X 0,Y 121.143,Z 700.546,A -85,B 0,C 180,E1 -27201.17,E2 -27201.17} C_VEL
LIN {X 0,Y 123.046,Z 697.696,A -85,B 0,C 180,E1 -27201.792,E2 -27201.792} C_VEL
LIN {X 0,Y 126.926,Z 693.136,A -85,B 0,C 180,E1 -27203.795,E2 -27203.795} C_VEL
LIN {X 0,Y 130.945,Z 687.33,A -85,B 0,C 180,E1 -27205.428,E2 -27205.428} C_VEL
LIN {X 0,Y 135.195,Z 679.481,A -85,B 0,C 180,E1 -27206.797,E2 -27206.797} C_VEL
LIN {X 0,Y 137.902,Z 673.384,A -85,B 0,C 180,E1 -27207.61,E2 -27207.61} C_VEL
LIN {X 0,Y 141.524,Z 667.584,A -85,B 0,C 180,E1 -27209.366,E2 -27209.366} C_VEL
LIN {X 0,Y 142.785,Z 666.661,A -85,B 0,C 180,E1 -27210.123,E2 -27210.123} C_VEL
LIN {X 0,Y 140.386,Z 680.063,A -85,B 0,C 180,E1 -27210.94,E2 -27210.94} C_VEL
LIN {X 0,Y 137,Z 692.921,A -85,B 0,C 180,E1 -27212.172,E2 -27212.172} C_VEL
LIN {X 0,Y 132.935,Z 704.172,A -85,B 0,C 180,E1 -27213.621,E2 -27213.621} C_VEL
LIN {X 0,Y 127.652,Z 715.786,A -85,B 0,C 180,E1 -27215.696,E2 -27215.696} C_VEL
LIN {X 0,Y 121.861,Z 726.224,A -85,B 0,C 180,E1 -27218.203,E2 -27218.203} C_VEL
LIN {X 0,Y 116.374,Z 734.747,A -85,B 0,C 180,E1 -27220.98,E2 -27220.98} C_VEL
LIN {X 0,Y 111.099,Z 741.995,A -85,B 0,C 180,E1 -27224.096,E2 -27224.096} C_VEL
LIN {X 0,Y 105.363,Z 749.1,A -85,B 0,C 180,E1 -27228.158,E2 -27228.158} C_VEL
LIN {X 0,Y 99.548,Z 755.503,A -85,B 0,C 180,E1 -27233.119,E2 -27233.119} C_VEL
LIN {X 0,Y 94.413,Z 760.583,A -85,B 0,C 180,E1 -27238.592,E2 -27238.592} C_VEL
LIN {X 0,Y 90.306,Z 764.518,A -85,B 0,C 180,E1 -27244.653,E2 -27244.653} C_VEL
LIN {X 0,Y 87.177,Z 767.421,A -85,B 0,C 180,E1 -27251.183,E2 -27251.183} C_VEL
LIN {X 0,Y 84.681,Z 769.791,A -85,B 0,C 180,E1 -27260.441,E2 -27260.441} C_VEL
LIN {X 0,Y 84.125,Z 770.395,A -85,B 0,C 180,E1 -27265.204,E2 -27265.204} C_VEL
LIN {X 0,Y 83.975,Z 770.619,A -85,B 0,C 180,E1 -27269.996,E2 -27269.996} C_VEL
LIN {X 0,Y 84.107,Z 770.424,A -85,B 0,C 180,E1 -27274.789,E2 -27274.789} C_VEL
LIN {X 0,Y 84.678,Z 769.84,A -85,B 0,C 180,E1 -27279.551,E2 -27279.551} C_VEL
LIN {X 0,Y 87.168,Z 767.517,A -85,B 0,C 180,E1 -27288.81,E2 -27288.81} C_VEL
LIN {X 0,Y 90.277,Z 764.645,A -85,B 0,C 180,E1 -27295.347,E2 -27295.347} C_VEL
LIN {X 0,Y 94.345,Z 760.749,A -85,B 0,C 180,E1 -27301.425,E2 -27301.425} C_VEL
LIN {X 0,Y 99.458,Z 755.721,A -85,B 0,C 180,E1 -27306.91,E2 -27306.91} C_VEL
LIN {X 0,Y 105.287,Z 749.387,A -85,B 0,C 180,E1 -27311.87,E2 -27311.87} C_VEL
LIN {X 0,Y 111.717,Z 741.434,A -85,B 0,C 180,E1 -27316.361,E2 -27316.361} C_VEL
LIN {X 0,Y 118.712,Z 731.605,A -85,B 0,C 180,E1 -27320.315,E2 -27320.315} C_VEL
LIN {X 0,Y 124.993,Z 721.24,A -85,B 0,C 180,E1 -27323.243,E2 -27323.243} C_VEL
LIN {X 0,Y 130.188,Z 710.98,A -85,B 0,C 180,E1 -27325.406,E2 -27325.406} C_VEL
LIN {X 0,Y 134.883,Z 699.735,A -85,B 0,C 180,E1 -27327.154,E2 -27327.154} C_VEL
LIN {X 0,Y 138.608,Z 688.286,A -85,B 0,C 180,E1 -27328.475,E2 -27328.475} C_VEL
LIN {X 0,Y 141.621,Z 675.483,A -85,B 0,C 180,E1 -27329.498,E2 -27329.498} C_VEL
LIN {X 0,Y 143.621,Z 661.88,A -85,B 0,C 180,E1 -27330.179,E2 -27330.179} C_VEL
LIN {X 0,Y 145.045,Z 646.28,A -85,B 0,C 180,E1 -27330.741,E2 -27330.741} C_VEL
LIN {X 0,Y 141.646,Z 638.734,A -85,B 0,C 180,E1 -27334.17,E2 -27334.17} C_VEL
LIN {X 0,Y 138.346,Z 632.233,A -85,B 0,C 180,E1 -27338.058,E2 -27338.058} C_VEL
LIN {X 0,Y 136.027,Z 628.242,A -85,B 0,C 180,E1 -27341.292,E2 -27341.292} C_VEL
LIN {X 0,Y 134.229,Z 625.061,A -85,B 0,C 180,E1 -27344.352,E2 -27344.352} C_VEL
LIN {X 0,Y 132.219,Z 621.363,A -85,B 0,C 180,E1 -27348.89,E2 -27348.89} C_VEL
LIN {X 0,Y 130.404,Z 616.625,A -85,B 0,C 180,E1 -27360,E2 -27360} C_VEL
LIN {X 0,Y 132.422,Z 621.709,A -85,B 0,C 180,E1 -27371.286,E2 -27371.286} C_VEL
LIN {X 0,Y 134.928,Z 626.284,A -85,B 0,C 180,E1 -27376.549,E2 -27376.549} C_VEL
LIN {X 0,Y 137.439,Z 630.671,A -85,B 0,C 180,E1 -27380.387,E2 -27380.387} C_VEL
LIN {X 0,Y 139.964,Z 635.425,A -85,B 0,C 180,E1 -27383.586,E2 -27383.586} C_VEL
LIN {X 0,Y 142.698,Z 643.022,A -85,B 0,C 180,E1 -27386.805,E2 -27386.805} C_VEL
LIN {X 0,Y 144.779,Z 649.594,A -85,B 0,C 180,E1 -27389.041,E2 -27389.041} C_VEL
LIN {X 0,Y 142.481,Z 672.162,A -85,B 0,C 180,E1 -27389.859,E2 -27389.859} C_VEL
LIN {X 0,Y 139.944,Z 685.487,A -85,B 0,C 180,E1 -27390.67,E2 -27390.67} C_VEL
LIN {X 0,Y 136.403,Z 697.936,A -85,B 0,C 180,E1 -27391.779,E2 -27391.779} C_VEL
LIN {X 0,Y 131.505,Z 710.587,A -85,B 0,C 180,E1 -27393.385,E2 -27393.385} C_VEL
LIN {X 0,Y 126.089,Z 721.838,A -85,B 0,C 180,E1 -27395.401,E2 -27395.401} C_VEL
LIN {X 0,Y 120.247,Z 731.973,A -85,B 0,C 180,E1 -27397.911,E2 -27397.911} C_VEL
LIN {X 0,Y 114.042,Z 741.113,A -85,B 0,C 180,E1 -27400.987,E2 -27400.987} C_VEL
LIN {X 0,Y 107.166,Z 750.028,A -85,B 0,C 180,E1 -27405.176,E2 -27405.176} C_VEL
LIN {X 0,Y 101.239,Z 756.98,A -85,B 0,C 180,E1 -27409.784,E2 -27409.784} C_VEL
LIN {X 0,Y 96.498,Z 762.052,A -85,B 0,C 180,E1 -27414.368,E2 -27414.368} C_VEL
LIN {X 0,Y 91.756,Z 766.764,A -85,B 0,C 180,E1 -27420.146,E2 -27420.146} C_VEL
LIN {X 0,Y 88.006,Z 770.37,A -85,B 0,C 180,E1 -27426.471,E2 -27426.471} C_VEL
LIN {X 0,Y 86.236,Z 772.233,A -85,B 0,C 180,E1 -27430.979,E2 -27430.979} C_VEL
LIN {X 0,Y 84.95,Z 773.631,A -85,B 0,C 180,E1 -27435.634,E2 -27435.634} C_VEL
LIN {X 0,Y 84.132,Z 774.632,A -85,B 0,C 180,E1 -27440.387,E2 -27440.387} C_VEL
LIN {X 0,Y 83.787,Z 775.243,A -85,B 0,C 180,E1 -27445.193,E2 -27445.193} C_VEL
LIN {X 0,Y 83.879,Z 775.459,A -85,B 0,C 180,E1 -27450.004,E2 -27450.004} C_VEL
LIN {X 0,Y 84.132,Z 775.234,A -85,B 0,C 180,E1 -27454.796,E2 -27454.796} C_VEL
LIN {X 0,Y 86.005,Z 773.615,A -85,B 0,C 180,E1 -27464.195,E2 -27464.195} C_VEL
LIN {X 0,Y 87.702,Z 772.21,A -85,B 0,C 180,E1 -27468.7,E2 -27468.7} C_VEL
LIN {X 0,Y 91.512,Z 769.283,A -85,B 0,C 180,E1 -27474.99,E2 -27474.99} C_VEL
LIN {X 0,Y 96.541,Z 765.325,A -85,B 0,C 180,E1 -27480.64,E2 -27480.64} C_VEL
LIN {X 0,Y 103.281,Z 760.2,A -85,B 0,C 180,E1 -27485.642,E2 -27485.642} C_VEL
LIN {X 0,Y 104.047,Z 760.401,A -85,B 0,C 180,E1 -27486.234,E2 -27486.234} C_VEL
LIN {X 0,Y 110.407,Z 766.412,A -85,B 0,C 180,E1 -27491.946,E2 -27491.946} C_VEL
LIN {X 0,Y 115.621,Z 769.934,A -85,B 0,C 180,E1 -27495.267,E2 -27495.267} C_VEL
LIN {X 0,Y 115.381,Z 769.736,A -85,B 0,C 180,E1 -27496.524,E2 -27496.524} C_VEL
LIN {X 0,Y 107.942,Z 763.916,A -85,B 0,C 180,E1 -27501.553,E2 -27501.553} C_VEL
LIN {X 0,Y 102.717,Z 757.64,A -85,B 0,C 180,E1 -27506.813,E2 -27506.813} C_VEL
LIN {X 0,Y 99.95,Z 752.614,A -85,B 0,C 180,E1 -27510.961,E2 -27510.961} C_VEL
LIN {X 0,Y 98.423,Z 750.121,A -85,B 0,C 180,E1 -27512.601,E2 -27512.601} C_VEL
LIN {X 0,Y 92.959,Z 744.522,A -85,B 0,C 180,E1 -27515.938,E2 -27515.938} C_VEL
LIN {X 0,Y 90.624,Z 742.309,A -85,B 0,C 180,E1 -27518.057,E2 -27518.057} C_VEL
LIN {X 0,Y 89.775,Z 741.219,A -85,B 0,C 180,E1 -27519.947,E2 -27519.947} C_VEL
LIN {X 0,Y 90.066,Z 739.291,A -85,B 0,C 180,E1 -27523.251,E2 -27523.251} C_VEL
LIN {X 0,Y 90.079,Z 737.856,A -85,B 0,C 180,E1 -27526.464,E2 -27526.464} C_VEL
LIN {X 0,Y 89.983,Z 736.373,A -85,B 0,C 180,E1 -27531.013,E2 -27531.013} C_VEL
LIN {X 0,Y 90.599,Z 735.145,A -85,B 0,C 180,E1 -27533.318,E2 -27533.318} C_VEL
LIN {X 0,Y 92.159,Z 732.521,A -85,B 0,C 180,E1 -27540,E2 -27540} C_VEL
LIN {X 0,Y 93.729,Z 730.771,A -85,B 0,C 180,E1 -27542.895,E2 -27542.895} C_VEL
LIN {X 0,Y 95.488,Z 729.156,A -85,B 0,C 180,E1 -27546.339,E2 -27546.339} C_VEL
LIN {X 0,Y 98.196,Z 726.598,A -85,B 0,C 180,E1 -27549.371,E2 -27549.371} C_VEL
LIN {X 0,Y 99.364,Z 725.508,A -85,B 0,C 180,E1 -27550.391,E2 -27550.391} C_VEL
LIN {X 0,Y 102.021,Z 723.413,A -85,B 0,C 180,E1 -27553.382,E2 -27553.382} C_VEL
LIN {X 0,Y 105.382,Z 720.424,A -85,B 0,C 180,E1 -27555.857,E2 -27555.857} C_VEL
LIN {X 0,Y 107.572,Z 718.297,A -85,B 0,C 180,E1 -27557.098,E2 -27557.098} C_VEL
LIN {X 0,Y 113.416,Z 713.174,A -85,B 0,C 180,E1 -27560.78,E2 -27560.78} C_VEL
LIN {X 0,Y 117.664,Z 708.892,A -85,B 0,C 180,E1 -27562.708,E2 -27562.708} C_VEL
LIN {X 0,Y 122.166,Z 703.437,A -85,B 0,C 180,E1 -27564.198,E2 -27564.198} C_VEL
LIN {X 0,Y 123.86,Z 701.329,A -85,B 0,C 180,E1 -27564.782,E2 -27564.782} C_VEL
LIN {X 0,Y 128.23,Z 696.44,A -85,B 0,C 180,E1 -27566.61,E2 -27566.61} C_VEL
LIN {X 0,Y 132.336,Z 690.984,A -85,B 0,C 180,E1 -27568.001,E2 -27568.001} C_VEL
LIN {X 0,Y 135.093,Z 686.586,A -85,B 0,C 180,E1 -27568.765,E2 -27568.765} C_VEL
LIN {X 0,Y 134.333,Z 689.992,A -85,B 0,C 180,E1 -27569.264,E2 -27569.264} C_VEL
LIN {X 0,Y 129.844,Z 702.659,A -85,B 0,C 180,E1 -27570.762,E2 -27570.762} C_VEL
LIN {X 0,Y 125.021,Z 713.374,A -85,B 0,C 180,E1 -27572.514,E2 -27572.514} C_VEL
LIN {X 0,Y 118.933,Z 724.3,A -85,B 0,C 180,E1 -27574.92,E2 -27574.92} C_VEL
LIN {X 0,Y 113.11,Z 733.179,A -85,B 0,C 180,E1 -27577.603,E2 -27577.603} C_VEL
LIN {X 0,Y 105.948,Z 742.628,A -85,B 0,C 180,E1 -27581.556,E2 -27581.556} C_VEL
LIN {X 0,Y 99.127,Z 750.469,A -85,B 0,C 180,E1 -27586.265,E2 -27586.265} C_VEL
LIN {X 0,Y 92.011,Z 757.517,A -85,B 0,C 180,E1 -27592.329,E2 -27592.329} C_VEL
LIN {X 0,Y 86.846,Z 762.203,A -85,B 0,C 180,E1 -27598.259,E2 -27598.259} C_VEL
LIN {X 0,Y 82.676,Z 765.78,A -85,B 0,C 180,E1 -27604.843,E2 -27604.843} C_VEL
LIN {X 0,Y 80.474,Z 767.627,A -85,B 0,C 180,E1 -27609.549,E2 -27609.549} C_VEL
LIN {X 0,Y 77.7,Z 769.996,A -85,B 0,C 180,E1 -27619.573,E2 -27619.573} C_VEL
LIN {X 0,Y 77.068,Z 770.599,A -85,B 0,C 180,E1 -27624.763,E2 -27624.763} C_VEL
LIN {X 0,Y 76.896,Z 770.823,A -85,B 0,C 180,E1 -27629.995,E2 -27629.995} C_VEL
LIN {X 0,Y 77.055,Z 770.628,A -85,B 0,C 180,E1 -27635.228,E2 -27635.228} C_VEL
LIN {X 0,Y 77.698,Z 770.044,A -85,B 0,C 180,E1 -27640.418,E2 -27640.418} C_VEL
LIN {X 0,Y 80.463,Z 767.722,A -85,B 0,C 180,E1 -27650.444,E2 -27650.444} C_VEL
LIN {X 0,Y 83.914,Z 764.849,A -85,B 0,C 180,E1 -27657.423,E2 -27657.423} C_VEL
LIN {X 0,Y 88.351,Z 760.953,A -85,B 0,C 180,E1 -27663.831,E2 -27663.831} C_VEL
LIN {X 0,Y 93.869,Z 755.925,A -85,B 0,C 180,E1 -27669.518,E2 -27669.518} C_VEL
LIN {X 0,Y 100.102,Z 749.59,A -85,B 0,C 180,E1 -27674.589,E2 -27674.589} C_VEL
LIN {X 0,Y 106.688,Z 741.961,A -85,B 0,C 180,E1 -27678.955,E2 -27678.955} C_VEL
LIN {X 0,Y 113.045,Z 733.585,A -85,B 0,C 180,E1 -27682.429,E2 -27682.429} C_VEL
LIN {X 0,Y 119.511,Z 723.72,A -85,B 0,C 180,E1 -27685.409,E2 -27685.409} C_VEL
LIN {X 0,Y 125.603,Z 712.602,A -85,B 0,C 180,E1 -27687.806,E2 -27687.806} C_VEL
LIN {X 0,Y 130.462,Z 701.698,A -85,B 0,C 180,E1 -27689.527,E2 -27689.527} C_VEL
LIN {X 0,Y 134.694,Z 689.629,A -85,B 0,C 180,E1 -27690.918,E2 -27690.918} C_VEL
LIN {X 0,Y 137.978,Z 676.643,A -85,B 0,C 180,E1 -27691.967,E2 -27691.967} C_VEL
LIN {X 0,Y 140.138,Z 662.9,A -85,B 0,C 180,E1 -27692.657,E2 -27692.657} C_VEL
LIN {X 0,Y 141.417,Z 649.476,A -85,B 0,C 180,E1 -27693.148,E2 -27693.148} C_VEL
LIN {X 0,Y 138.474,Z 642.731,A -85,B 0,C 180,E1 -27696.537,E2 -27696.537} C_VEL
LIN {X 0,Y 135.553,Z 636.838,A -85,B 0,C 180,E1 -27700.502,E2 -27700.502} C_VEL
LIN {X 0,Y 132.919,Z 631.843,A -85,B 0,C 180,E1 -27705.062,E2 -27705.062} C_VEL
LIN {X 0,Y 131.069,Z 628.22,A -85,B 0,C 180,E1 -27709.574,E2 -27709.574} C_VEL
LIN {X 0,Y 129.528,Z 623.759,A -85,B 0,C 180,E1 -27720,E2 -27720} C_VEL
LIN {X 0,Y 131.25,Z 628.616,A -85,B 0,C 180,E1 -27730.607,E2 -27730.607} C_VEL
LIN {X 0,Y 133.423,Z 632.86,A -85,B 0,C 180,E1 -27735.576,E2 -27735.576} C_VEL
LIN {X 0,Y 135.683,Z 637.071,A -85,B 0,C 180,E1 -27739.33,E2 -27739.33} C_VEL
LIN {X 0,Y 137.874,Z 641.69,A -85,B 0,C 180,E1 -27742.378,E2 -27742.378} C_VEL
LIN {X 0,Y 140.386,Z 649.47,A -85,B 0,C 180,E1 -27745.641,E2 -27745.641} C_VEL
LIN {X 0,Y 141.187,Z 652.267,A -85,B 0,C 180,E1 -27746.615,E2 -27746.615} C_VEL
LIN {X 0,Y 139.08,Z 671.887,A -85,B 0,C 180,E1 -27747.305,E2 -27747.305} C_VEL
LIN {X 0,Y 136.411,Z 685.506,A -85,B 0,C 180,E1 -27748.122,E2 -27748.122} C_VEL
LIN {X 0,Y 132.802,Z 697.737,A -85,B 0,C 180,E1 -27749.174,E2 -27749.174} C_VEL
LIN {X 0,Y 127.738,Z 710.387,A -85,B 0,C 180,E1 -27750.727,E2 -27750.727} C_VEL
LIN {X 0,Y 122.115,Z 721.637,A -85,B 0,C 180,E1 -27752.686,E2 -27752.686} C_VEL
LIN {X 0,Y 116.01,Z 731.771,A -85,B 0,C 180,E1 -27755.137,E2 -27755.137} C_VEL
LIN {X 0,Y 109.517,Z 740.911,A -85,B 0,C 180,E1 -27758.182,E2 -27758.182} C_VEL
LIN {X 0,Y 102.236,Z 749.824,A -85,B 0,C 180,E1 -27762.361,E2 -27762.361} C_VEL
LIN {X 0,Y 95.371,Z 757.316,A -85,B 0,C 180,E1 -27767.469,E2 -27767.469} C_VEL
LIN {X 0,Y 90.813,Z 761.849,A -85,B 0,C 180,E1 -27771.754,E2 -27771.754} C_VEL
LIN {X 0,Y 85.645,Z 766.559,A -85,B 0,C 180,E1 -27777.771,E2 -27777.771} C_VEL
LIN {X 0,Y 81.512,Z 770.165,A -85,B 0,C 180,E1 -27784.467,E2 -27784.467} C_VEL
LIN {X 0,Y 79.519,Z 772.028,A -85,B 0,C 180,E1 -27789.302,E2 -27789.302} C_VEL
LIN {X 0,Y 78.055,Z 773.426,A -85,B 0,C 180,E1 -27794.334,E2 -27794.334} C_VEL
LIN {X 0,Y 77.119,Z 774.427,A -85,B 0,C 180,E1 -27799.503,E2 -27799.503} C_VEL
LIN {X 0,Y 76.707,Z 775.039,A -85,B 0,C 180,E1 -27804.748,E2 -27804.748} C_VEL
LIN {X 0,Y 76.777,Z 775.255,A -85,B 0,C 180,E1 -27810.005,E2 -27810.005} C_VEL
LIN {X 0,Y 77.076,Z 775.03,A -85,B 0,C 180,E1 -27815.236,E2 -27815.236} C_VEL
LIN {X 0,Y 79.137,Z 773.41,A -85,B 0,C 180,E1 -27825.456,E2 -27825.456} C_VEL
LIN {X 0,Y 81.02,Z 772.005,A -85,B 0,C 180,E1 -27830.307,E2 -27830.307} C_VEL
LIN {X 0,Y 85.138,Z 769.078,A -85,B 0,C 180,E1 -27837.006,E2 -27837.006} C_VEL
LIN {X 0,Y 90.517,Z 765.123,A -85,B 0,C 180,E1 -27842.927,E2 -27842.927} C_VEL
LIN {X 0,Y 98.508,Z 759.066,A -85,B 0,C 180,E1 -27848.632,E2 -27848.632} C_VEL
LIN {X 0,Y 100.141,Z 758.151,A -85,B 0,C 180,E1 -27849.5,E2 -27849.5} C_VEL
LIN {X 0,Y 100.948,Z 758.5,A -85,B 0,C 180,E1 -27850.094,E2 -27850.094} C_VEL
LIN {X 0,Y 108.003,Z 764.734,A -85,B 0,C 180,E1 -27855.713,E2 -27855.713} C_VEL
LIN {X 0,Y 101.043,Z 758.085,A -85,B 0,C 180,E1 -27861.245,E2 -27861.245} C_VEL
LIN {X 0,Y 95.304,Z 749.152,A -85,B 0,C 180,E1 -27868.556,E2 -27868.556} C_VEL
LIN {X 0,Y 92.965,Z 743.752,A -85,B 0,C 180,E1 -27873.026,E2 -27873.026} C_VEL
LIN {X 0,Y 91.731,Z 742.69,A -85,B 0,C 180,E1 -27874.775,E2 -27874.775} C_VEL
LIN {X 0,Y 90.331,Z 742.32,A -85,B 0,C 180,E1 -27877.107,E2 -27877.107} C_VEL
LIN {X 0,Y 89.775,Z 741.219,A -85,B 0,C 180,E1 -27879.947,E2 -27879.947} C_VEL
LIN {X 0,Y 88.977,Z 740.678,A -85,B 0,C 180,E1 -27882.437,E2 -27882.437} C_VEL
LIN {X 0,Y 85.118,Z 740.967,A -85,B 0,C 180,E1 -27890.958,E2 -27890.958} C_VEL
LIN {X 0,Y 85.192,Z 740.288,A -85,B 0,C 180,E1 -27893.587,E2 -27893.587} C_VEL
LIN {X 0,Y 87.898,Z 736.903,A -85,B 0,C 180,E1 -27902.291,E2 -27902.291} C_VEL
LIN {X 0,Y 89.226,Z 735.665,A -85,B 0,C 180,E1 -27904.518,E2 -27904.518} C_VEL
LIN {X 0,Y 91.801,Z 733.665,A -85,B 0,C 180,E1 -27908.808,E2 -27908.808} C_VEL
LIN {X 0,Y 94.59,Z 731.435,A -85,B 0,C 180,E1 -27911.682,E2 -27911.682} C_VEL
LIN {X 0,Y 95.874,Z 730.384,A -85,B 0,C 180,E1 -27912.704,E2 -27912.704} C_VEL
LIN {X 0,Y 99.741,Z 727.688,A -85,B 0,C 180,E1 -27916.371,E2 -27916.371} C_VEL
LIN {X 0,Y 104.117,Z 724.226,A -85,B 0,C 180,E1 -27919.08,E2 -27919.08} C_VEL
LIN {X 0,Y 107.687,Z 721.31,A -85,B 0,C 180,E1 -27921.061,E2 -27921.061} C_VEL
LIN {X 0,Y 113.031,Z 717.046,A -85,B 0,C 180,E1 -27923.838,E2 -27923.838} C_VEL
LIN {X 0,Y 117.295,Z 713.12,A -85,B 0,C 180,E1 -27925.481,E2 -27925.481} C_VEL
LIN {X 0,Y 124.357,Z 705.372,A -85,B 0,C 180,E1 -27927.51,E2 -27927.51} C_VEL
LIN {X 0,Y 125.373,Z 704.412,A -85,B 0,C 180,E1 -27927.895,E2 -27927.895} C_VEL
LIN {X 0,Y 124.942,Z 706.165,A -85,B 0,C 180,E1 -27928.481,E2 -27928.481} C_VEL
LIN {X 0,Y 119.226,Z 717.492,A -85,B 0,C 180,E1 -27930.442,E2 -27930.442} C_VEL
LIN {X 0,Y 112.957,Z 727.693,A -85,B 0,C 180,E1 -27932.86,E2 -27932.86} C_VEL
LIN {X 0,Y 106.3,Z 736.845,A -85,B 0,C 180,E1 -27935.908,E2 -27935.908} C_VEL
LIN {X 0,Y 98.78,Z 745.761,A -85,B 0,C 180,E1 -27940.127,E2 -27940.127} C_VEL
LIN {X 0,Y 91.871,Z 752.895,A -85,B 0,C 180,E1 -27944.954,E2 -27944.954} C_VEL
LIN {X 0,Y 86.514,Z 757.722,A -85,B 0,C 180,E1 -27949.462,E2 -27949.462} C_VEL
LIN {X 0,Y 80.886,Z 762.409,A -85,B 0,C 180,E1 -27955.609,E2 -27955.609} C_VEL
LIN {X 0,Y 76.307,Z 765.986,A -85,B 0,C 180,E1 -27962.575,E2 -27962.575} C_VEL
LIN {X 0,Y 73.858,Z 767.832,A -85,B 0,C 180,E1 -27967.623,E2 -27967.623} C_VEL
LIN {X 0,Y 72.008,Z 769.216,A -85,B 0,C 180,E1 -27972.969,E2 -27972.969} C_VEL
LIN {X 0,Y 70.008,Z 770.804,A -85,B 0,C 180,E1 -27984.233,E2 -27984.233} C_VEL
LIN {X 0,Y 69.815,Z 771.027,A -85,B 0,C 180,E1 -27989.995,E2 -27989.995} C_VEL
LIN {X 0,Y 69.999,Z 770.832,A -85,B 0,C 180,E1 -27995.757,E2 -27995.757} C_VEL
LIN {X 0,Y 72.003,Z 769.283,A -85,B 0,C 180,E1 -28007.022,E2 -28007.022} C_VEL
LIN {X 0,Y 73.845,Z 767.926,A -85,B 0,C 180,E1 -28012.371,E2 -28012.371} C_VEL
LIN {X 0,Y 77.666,Z 765.054,A -85,B 0,C 180,E1 -28019.842,E2 -28019.842} C_VEL
LIN {X 0,Y 82.536,Z 761.157,A -85,B 0,C 180,E1 -28026.582,E2 -28026.582} C_VEL
LIN {X 0,Y 88.505,Z 756.128,A -85,B 0,C 180,E1 -28032.445,E2 -28032.445} C_VEL
LIN {X 0,Y 95.169,Z 749.793,A -85,B 0,C 180,E1 -28037.596,E2 -28037.596} C_VEL
LIN {X 0,Y 102.408,Z 741.871,A -85,B 0,C 180,E1 -28042.103,E2 -28042.103} C_VEL
LIN {X 0,Y 108.854,Z 733.787,A -85,B 0,C 180,E1 -28045.398,E2 -28045.398} C_VEL
LIN {X 0,Y 115.634,Z 723.921,A -85,B 0,C 180,E1 -28048.302,E2 -28048.302} C_VEL
LIN {X 0,Y 121.976,Z 712.802,A -85,B 0,C 180,E1 -28050.623,E2 -28050.623} C_VEL
LIN {X 0,Y 127.01,Z 701.897,A -85,B 0,C 180,E1 -28052.287,E2 -28052.287} C_VEL
LIN {X 0,Y 131.396,Z 689.826,A -85,B 0,C 180,E1 -28053.618,E2 -28053.618} C_VEL
LIN {X 0,Y 134.664,Z 677.47,A -85,B 0,C 180,E1 -28054.59,E2 -28054.59} C_VEL
LIN {X 0,Y 136.904,Z 664.065,A -85,B 0,C 180,E1 -28055.259,E2 -28055.259} C_VEL
LIN {X 0,Y 138.027,Z 652.807,A -85,B 0,C 180,E1 -28055.683,E2 -28055.683} C_VEL
LIN {X 0,Y 135.515,Z 646.814,A -85,B 0,C 180,E1 -28059.036,E2 -28059.036} C_VEL
LIN {X 0,Y 133.083,Z 641.619,A -85,B 0,C 180,E1 -28062.917,E2 -28062.917} C_VEL
LIN {X 0,Y 131.231,Z 638.001,A -85,B 0,C 180,E1 -28066.647,E2 -28066.647} C_VEL
LIN {X 0,Y 129.814,Z 634.921,A -85,B 0,C 180,E1 -28070.653,E2 -28070.653} C_VEL
LIN {X 0,Y 128.64,Z 630.987,A -85,B 0,C 180,E1 -28080,E2 -28080} C_VEL
LIN {X 0,Y 130.101,Z 635.487,A -85,B 0,C 180,E1 -28089.915,E2 -28089.915} C_VEL
LIN {X 0,Y 131.994,Z 639.478,A -85,B 0,C 180,E1 -28094.65,E2 -28094.65} C_VEL
LIN {X 0,Y 133.864,Z 643.242,A -85,B 0,C 180,E1 -28098.064,E2 -28098.064} C_VEL
LIN {X 0,Y 135.668,Z 647.435,A -85,B 0,C 180,E1 -28100.864,E2 -28100.864} C_VEL
LIN {X 0,Y 137.797,Z 654.717,A -85,B 0,C 180,E1 -28103.981,E2 -28103.981} C_VEL
LIN {X 0,Y 137.562,Z 658.104,A -85,B 0,C 180,E1 -28104.185,E2 -28104.185} C_VEL
LIN {X 0,Y 135.567,Z 674.323,A -85,B 0,C 180,E1 -28104.787,E2 -28104.787} C_VEL
LIN {X 0,Y 132.726,Z 687.222,A -85,B 0,C 180,E1 -28105.567,E2 -28105.567} C_VEL
LIN {X 0,Y 128.742,Z 699.536,A -85,B 0,C 180,E1 -28106.638,E2 -28106.638} C_VEL
LIN {X 0,Y 123.531,Z 711.772,A -85,B 0,C 180,E1 -28108.142,E2 -28108.142} C_VEL
LIN {X 0,Y 117.706,Z 722.679,A -85,B 0,C 180,E1 -28110.037,E2 -28110.037} C_VEL
LIN {X 0,Y 110.685,Z 733.525,A -85,B 0,C 180,E1 -28112.728,E2 -28112.728} C_VEL
